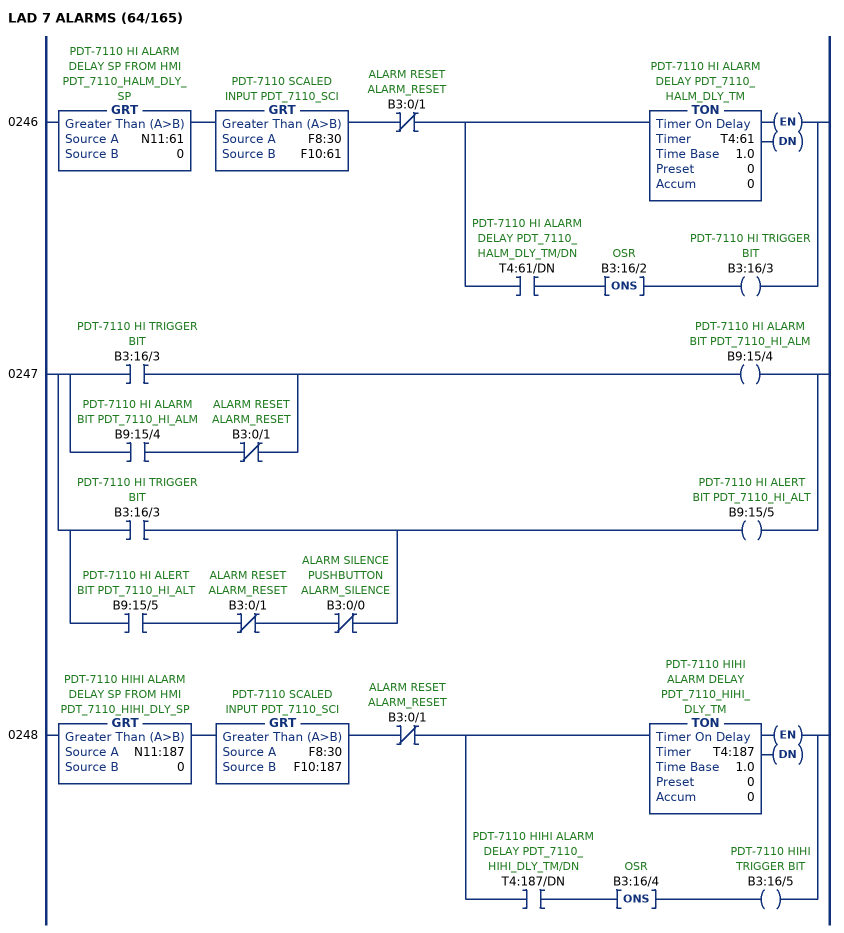
% Rung: 246 %
SOR GRT N11:61 0 GRT F8:30 F10:61 XIO B3:0/1 BST TON T4:61 1.0 0 0 NXB XIC T4:61/DN OSR B3:16/2 OTE B3:16/3 BND EOR
%   N11:61  PDT_7110_HALM_DLY_SP  "PDT-7110 HI ALARM DELAY SP FROM HMI" %
%   F8:30  PDT_7110_SCI  "PDT-7110 SCALED INPUT" %
%   F10:61  PDT_7110_HIALM_SP  "PDT-7110 HI ALARM SP" %
%   B3:0/1  ALARM_RESET  "ALARM RESET" %
%   T4:61  PDT_7110_HALM_DLY_TM  "PDT-7110 HI ALARM DELAY" %
%   B3:16/2  "OSR" %
%   B3:16/3  "PDT-7110 HI TRIGGER BIT" %
% Rung: 247 %
SOR BST BST XIC B3:16/3 NXB XIC B9:15/4 XIO B3:0/1 BND OTE B9:15/4 NXB BST XIC B3:16/3 NXB XIC B9:15/5 XIO B3:0/1 XIO B3:0/0 BND OTE B9:15/5 BND EOR
%   B3:16/3  "PDT-7110 HI TRIGGER BIT" %
%   B9:15/4  PDT_7110_HI_ALM  "PDT-7110 HI ALARM BIT" %
%   B3:0/1  ALARM_RESET  "ALARM RESET" %
%   B9:15/5  PDT_7110_HI_ALT  "PDT-7110 HI ALERT BIT" %
%   B3:0/0  ALARM_SILENCE  "ALARM SILENCE PUSHBUTTON" %
% Rung: 248 %
SOR GRT N11:187 0 GRT F8:30 F10:187 XIO B3:0/1 BST TON T4:187 1.0 0 0 NXB XIC T4:187/DN OSR B3:16/4 OTE B3:16/5 BND EOR
%   N11:187  PDT_7110_HIHI_DLY_SP  "PDT-7110 HIHI ALARM DELAY SP FROM HMI" %
%   F8:30  PDT_7110_SCI  "PDT-7110 SCALED INPUT" %
%   F10:187  PDT_7110_HIHI_SP  "PDT-7110 HIHI ALARM SP" %
%   B3:0/1  ALARM_RESET  "ALARM RESET" %
%   T4:187  PDT_7110_HIHI_DLY_TM  "PDT-7110 HIHI ALARM DELAY" %
%   B3:16/4  "OSR" %
%   B3:16/5  "PDT-7110 HIHI TRIGGER BIT" %

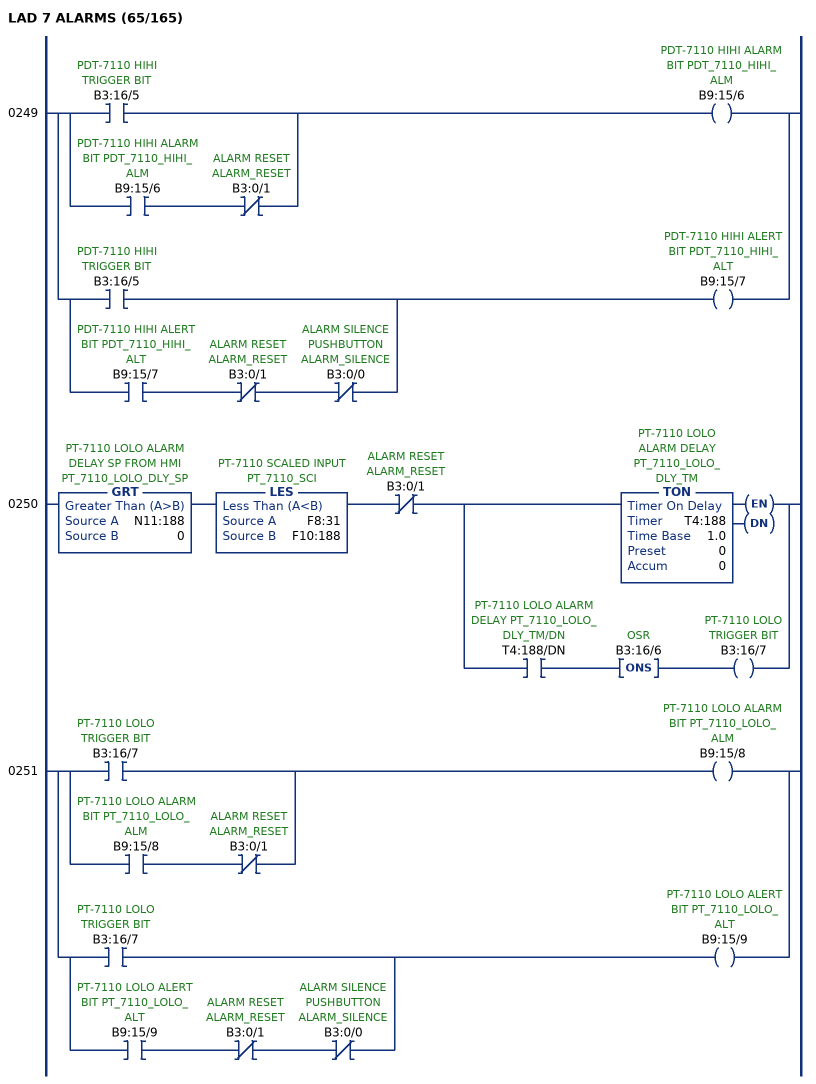
% Rung: 249 %
SOR BST BST XIC B3:16/5 NXB XIC B9:15/6 XIO B3:0/1 BND OTE B9:15/6 NXB BST XIC B3:16/5 NXB XIC B9:15/7 XIO B3:0/1 XIO B3:0/0 BND OTE B9:15/7 BND EOR
%   B3:16/5  "PDT-7110 HIHI TRIGGER BIT" %
%   B9:15/6  PDT_7110_HIHI_ALM  "PDT-7110 HIHI ALARM BIT" %
%   B3:0/1  ALARM_RESET  "ALARM RESET" %
%   B9:15/7  PDT_7110_HIHI_ALT  "PDT-7110 HIHI ALERT BIT" %
%   B3:0/0  ALARM_SILENCE  "ALARM SILENCE PUSHBUTTON" %
% Rung: 250 %
SOR GRT N11:188 0 LES F8:31 F10:188 XIO B3:0/1 BST TON T4:188 1.0 0 0 NXB XIC T4:188/DN OSR B3:16/6 OTE B3:16/7 BND EOR
%   N11:188  PT_7110_LOLO_DLY_SP  "PT-7110 LOLO ALARM DELAY SP FROM HMI" %
%   F8:31  PT_7110_SCI  "PT-7110 SCALED INPUT" %
%   F10:188  PT_7110_LOLO_SP  "PT-7110 LOLO ALARM SP" %
%   B3:0/1  ALARM_RESET  "ALARM RESET" %
%   T4:188  PT_7110_LOLO_DLY_TM  "PT-7110 LOLO ALARM DELAY" %
%   B3:16/6  "OSR" %
%   B3:16/7  "PT-7110 LOLO TRIGGER BIT" %
% Rung: 251 %
SOR BST BST XIC B3:16/7 NXB XIC B9:15/8 XIO B3:0/1 BND OTE B9:15/8 NXB BST XIC B3:16/7 NXB XIC B9:15/9 XIO B3:0/1 XIO B3:0/0 BND OTE B9:15/9 BND EOR
%   B3:16/7  "PT-7110 LOLO TRIGGER BIT" %
%   B9:15/8  PT_7110_LOLO_ALM  "PT-7110 LOLO ALARM BIT" %
%   B3:0/1  ALARM_RESET  "ALARM RESET" %
%   B9:15/9  PT_7110_LOLO_ALT  "PT-7110 LOLO ALERT BIT" %
%   B3:0/0  ALARM_SILENCE  "ALARM SILENCE PUSHBUTTON" %

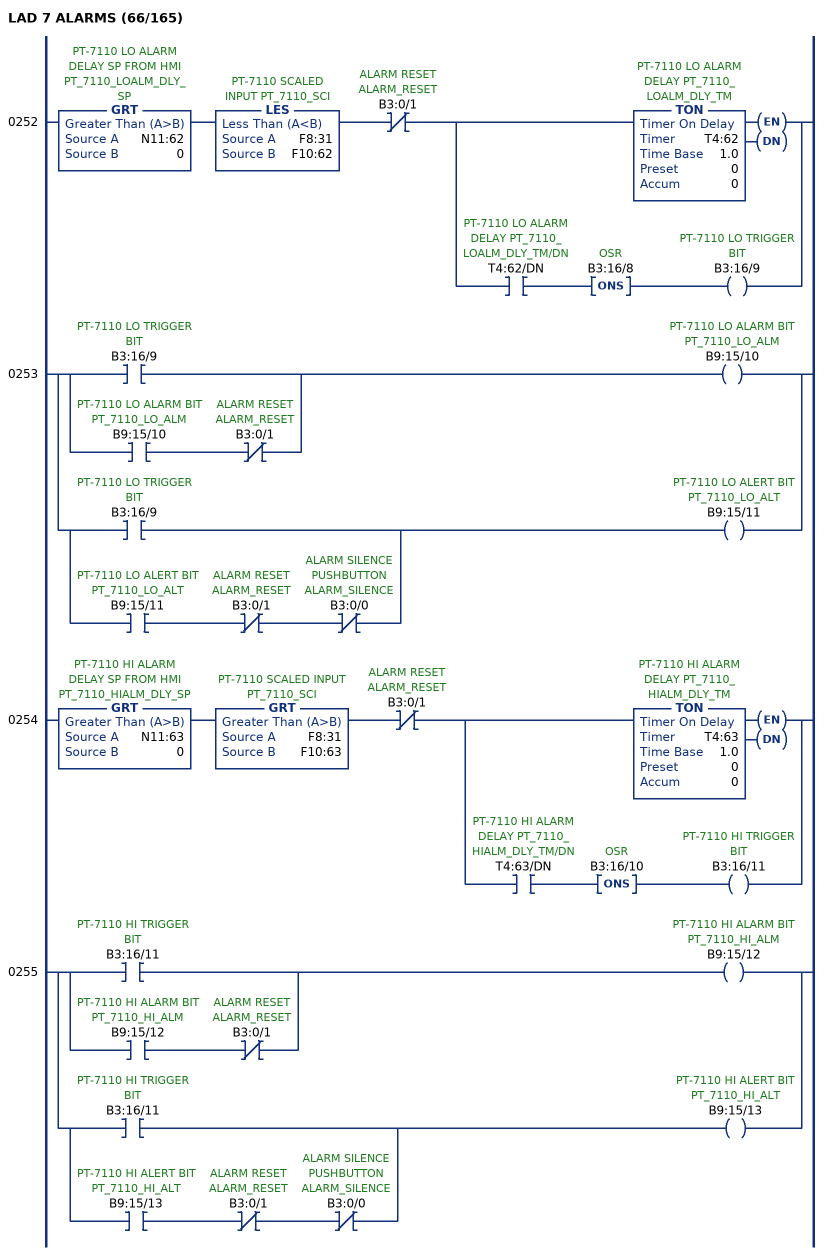
% Rung: 252 %
SOR GRT N11:62 0 LES F8:31 F10:62 XIO B3:0/1 BST TON T4:62 1.0 0 0 NXB XIC T4:62/DN OSR B3:16/8 OTE B3:16/9 BND EOR
%   N11:62  PT_7110_LOALM_DLY_SP  "PT-7110 LO ALARM DELAY SP FROM HMI" %
%   F8:31  PT_7110_SCI  "PT-7110 SCALED INPUT" %
%   F10:62  PT_7110_LOALM_SP  "PT-7110 LO ALARM SP" %
%   B3:0/1  ALARM_RESET  "ALARM RESET" %
%   T4:62  PT_7110_LOALM_DLY_TM  "PT-7110 LO ALARM DELAY" %
%   B3:16/8  "OSR" %
%   B3:16/9  "PT-7110 LO TRIGGER BIT" %
% Rung: 253 %
SOR BST BST XIC B3:16/9 NXB XIC B9:15/10 XIO B3:0/1 BND OTE B9:15/10 NXB BST XIC B3:16/9 NXB XIC B9:15/11 XIO B3:0/1 XIO B3:0/0 BND OTE B9:15/11 BND EOR
%   B3:16/9  "PT-7110 LO TRIGGER BIT" %
%   B9:15/10  PT_7110_LO_ALM  "PT-7110 LO ALARM BIT" %
%   B3:0/1  ALARM_RESET  "ALARM RESET" %
%   B9:15/11  PT_7110_LO_ALT  "PT-7110 LO ALERT BIT" %
%   B3:0/0  ALARM_SILENCE  "ALARM SILENCE PUSHBUTTON" %
% Rung: 254 %
SOR GRT N11:63 0 GRT F8:31 F10:63 XIO B3:0/1 BST TON T4:63 1.0 0 0 NXB XIC T4:63/DN OSR B3:16/10 OTE B3:16/11 BND EOR
%   N11:63  PT_7110_HIALM_DLY_SP  "PT-7110 HI ALARM DELAY SP FROM HMI" %
%   F8:31  PT_7110_SCI  "PT-7110 SCALED INPUT" %
%   F10:63  PT_7110_HIALM_SP  "PT-7110 HI ALARM SP" %
%   B3:0/1  ALARM_RESET  "ALARM RESET" %
%   T4:63  PT_7110_HIALM_DLY_TM  "PT-7110 HI ALARM DELAY" %
%   B3:16/10  "OSR" %
%   B3:16/11  "PT-7110 HI TRIGGER BIT" %
% Rung: 255 %
SOR BST BST XIC B3:16/11 NXB XIC B9:15/12 XIO B3:0/1 BND OTE B9:15/12 NXB BST XIC B3:16/11 NXB XIC B9:15/13 XIO B3:0/1 XIO B3:0/0 BND OTE B9:15/13 BND EOR
%   B3:16/11  "PT-7110 HI TRIGGER BIT" %
%   B9:15/12  PT_7110_HI_ALM  "PT-7110 HI ALARM BIT" %
%   B3:0/1  ALARM_RESET  "ALARM RESET" %
%   B9:15/13  PT_7110_HI_ALT  "PT-7110 HI ALERT BIT" %
%   B3:0/0  ALARM_SILENCE  "ALARM SILENCE PUSHBUTTON" %

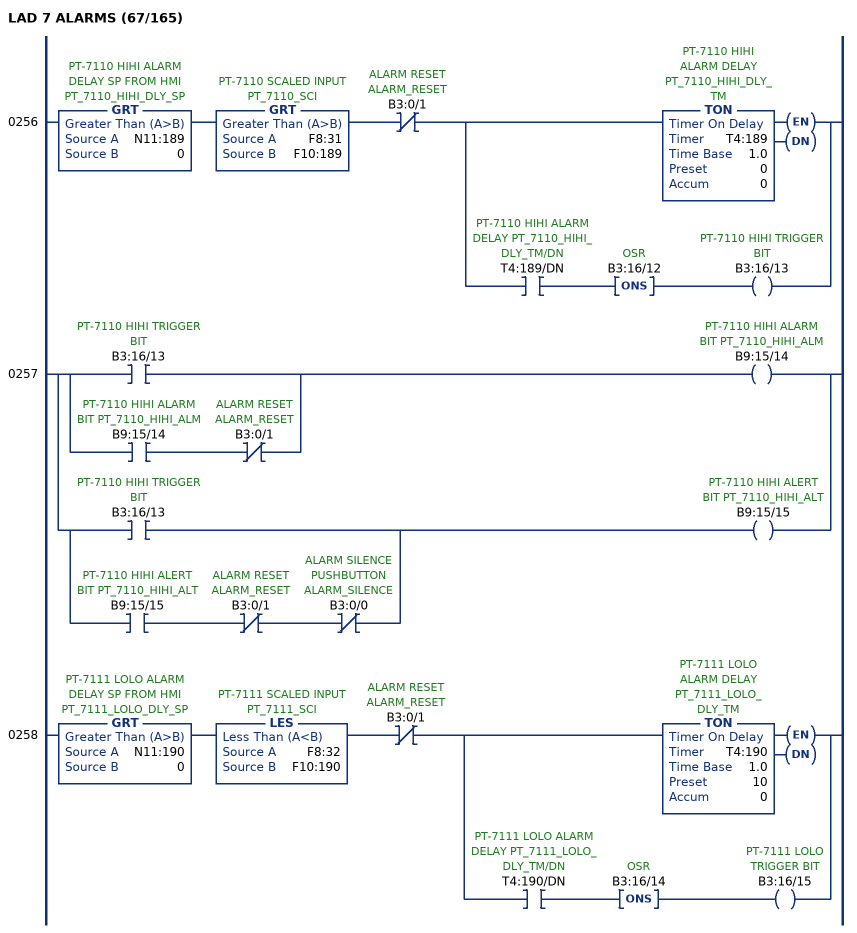
% Rung: 256 %
SOR GRT N11:189 0 GRT F8:31 F10:189 XIO B3:0/1 BST TON T4:189 1.0 0 0 NXB XIC T4:189/DN OSR B3:16/12 OTE B3:16/13 BND EOR
%   N11:189  PT_7110_HIHI_DLY_SP  "PT-7110 HIHI ALARM DELAY SP FROM HMI" %
%   F8:31  PT_7110_SCI  "PT-7110 SCALED INPUT" %
%   F10:189  PT_7110_HIHI_SP  "PT-7110 HIHI ALARM SP" %
%   B3:0/1  ALARM_RESET  "ALARM RESET" %
%   T4:189  PT_7110_HIHI_DLY_TM  "PT-7110 HIHI ALARM DELAY" %
%   B3:16/12  "OSR" %
%   B3:16/13  "PT-7110 HIHI TRIGGER BIT" %
% Rung: 257 %
SOR BST BST XIC B3:16/13 NXB XIC B9:15/14 XIO B3:0/1 BND OTE B9:15/14 NXB BST XIC B3:16/13 NXB XIC B9:15/15 XIO B3:0/1 XIO B3:0/0 BND OTE B9:15/15 BND EOR
%   B3:16/13  "PT-7110 HIHI TRIGGER BIT" %
%   B9:15/14  PT_7110_HIHI_ALM  "PT-7110 HIHI ALARM BIT" %
%   B3:0/1  ALARM_RESET  "ALARM RESET" %
%   B9:15/15  PT_7110_HIHI_ALT  "PT-7110 HIHI ALERT BIT" %
%   B3:0/0  ALARM_SILENCE  "ALARM SILENCE PUSHBUTTON" %
% Rung: 258 %
SOR GRT N11:190 0 LES F8:32 F10:190 XIO B3:0/1 BST TON T4:190 1.0 10 0 NXB XIC T4:190/DN OSR B3:16/14 OTE B3:16/15 BND EOR
%   N11:190  PT_7111_LOLO_DLY_SP  "PT-7111 LOLO ALARM DELAY SP FROM HMI" %
%   F8:32  PT_7111_SCI  "PT-7111 SCALED INPUT" %
%   F10:190  PT_7111_LOLO_SP  "PT-7111 LOLO ALARM SP" %
%   B3:0/1  ALARM_RESET  "ALARM RESET" %
%   T4:190  PT_7111_LOLO_DLY_TM  "PT-7111 LOLO ALARM DELAY" %
%   B3:16/14  "OSR" %
%   B3:16/15  "PT-7111 LOLO TRIGGER BIT" %

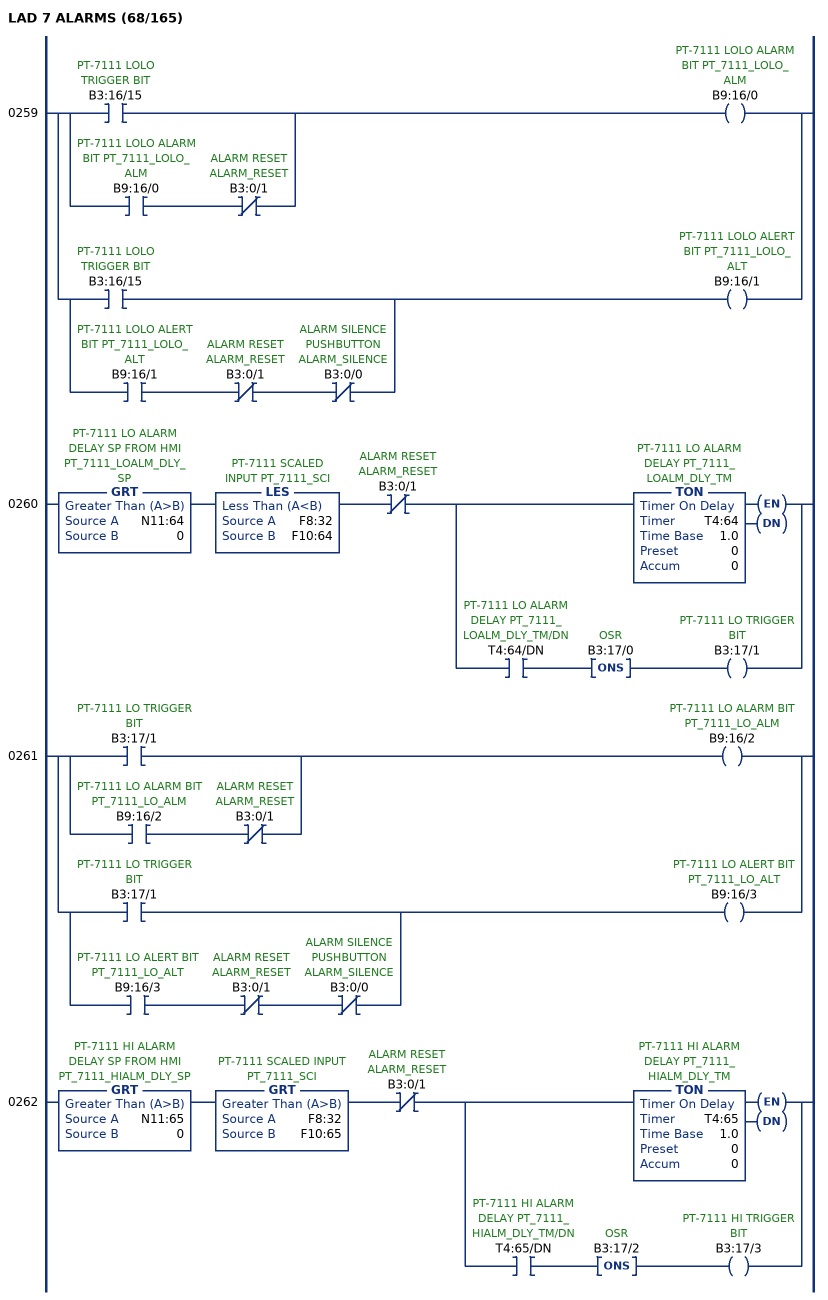
% Rung: 259 %
SOR BST BST XIC B3:16/15 NXB XIC B9:16/0 XIO B3:0/1 BND OTE B9:16/0 NXB BST XIC B3:16/15 NXB XIC B9:16/1 XIO B3:0/1 XIO B3:0/0 BND OTE B9:16/1 BND EOR
%   B3:16/15  "PT-7111 LOLO TRIGGER BIT" %
%   B9:16/0  PT_7111_LOLO_ALM  "PT-7111 LOLO ALARM BIT" %
%   B3:0/1  ALARM_RESET  "ALARM RESET" %
%   B9:16/1  PT_7111_LOLO_ALT  "PT-7111 LOLO ALERT BIT" %
%   B3:0/0  ALARM_SILENCE  "ALARM SILENCE PUSHBUTTON" %
% Rung: 260 %
SOR GRT N11:64 0 LES F8:32 F10:64 XIO B3:0/1 BST TON T4:64 1.0 0 0 NXB XIC T4:64/DN OSR B3:17/0 OTE B3:17/1 BND EOR
%   N11:64  PT_7111_LOALM_DLY_SP  "PT-7111 LO ALARM DELAY SP FROM HMI" %
%   F8:32  PT_7111_SCI  "PT-7111 SCALED INPUT" %
%   F10:64  PT_7111_LOALM_SP  "PT-7111 LO ALARM SP" %
%   B3:0/1  ALARM_RESET  "ALARM RESET" %
%   T4:64  PT_7111_LOALM_DLY_TM  "PT-7111 LO ALARM DELAY" %
%   B3:17/0  "OSR" %
%   B3:17/1  "PT-7111 LO TRIGGER BIT" %
% Rung: 261 %
SOR BST BST XIC B3:17/1 NXB XIC B9:16/2 XIO B3:0/1 BND OTE B9:16/2 NXB BST XIC B3:17/1 NXB XIC B9:16/3 XIO B3:0/1 XIO B3:0/0 BND OTE B9:16/3 BND EOR
%   B3:17/1  "PT-7111 LO TRIGGER BIT" %
%   B9:16/2  PT_7111_LO_ALM  "PT-7111 LO ALARM BIT" %
%   B3:0/1  ALARM_RESET  "ALARM RESET" %
%   B9:16/3  PT_7111_LO_ALT  "PT-7111 LO ALERT BIT" %
%   B3:0/0  ALARM_SILENCE  "ALARM SILENCE PUSHBUTTON" %
% Rung: 262 %
SOR GRT N11:65 0 GRT F8:32 F10:65 XIO B3:0/1 BST TON T4:65 1.0 0 0 NXB XIC T4:65/DN OSR B3:17/2 OTE B3:17/3 BND EOR
%   N11:65  PT_7111_HIALM_DLY_SP  "PT-7111 HI ALARM DELAY SP FROM HMI" %
%   F8:32  PT_7111_SCI  "PT-7111 SCALED INPUT" %
%   F10:65  PT_7111_HIALM_SP  "PT-7111 HI ALARM SP" %
%   B3:0/1  ALARM_RESET  "ALARM RESET" %
%   T4:65  PT_7111_HIALM_DLY_TM  "PT-7111 HI ALARM DELAY" %
%   B3:17/2  "OSR" %
%   B3:17/3  "PT-7111 HI TRIGGER BIT" %

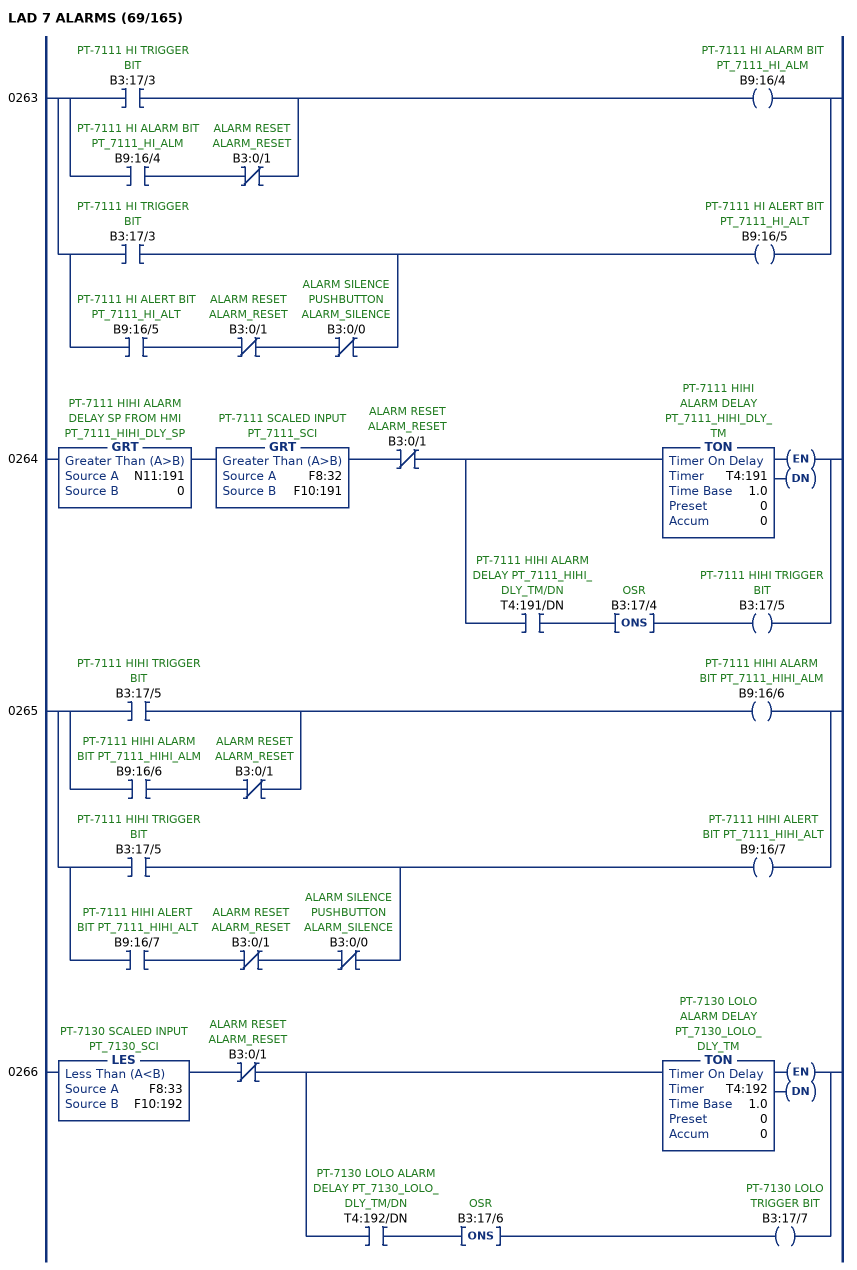
% Rung: 263 %
SOR BST BST XIC B3:17/3 NXB XIC B9:16/4 XIO B3:0/1 BND OTE B9:16/4 NXB BST XIC B3:17/3 NXB XIC B9:16/5 XIO B3:0/1 XIO B3:0/0 BND OTE B9:16/5 BND EOR
%   B3:17/3  "PT-7111 HI TRIGGER BIT" %
%   B9:16/4  PT_7111_HI_ALM  "PT-7111 HI ALARM BIT" %
%   B3:0/1  ALARM_RESET  "ALARM RESET" %
%   B9:16/5  PT_7111_HI_ALT  "PT-7111 HI ALERT BIT" %
%   B3:0/0  ALARM_SILENCE  "ALARM SILENCE PUSHBUTTON" %
% Rung: 264 %
SOR GRT N11:191 0 GRT F8:32 F10:191 XIO B3:0/1 BST TON T4:191 1.0 0 0 NXB XIC T4:191/DN OSR B3:17/4 OTE B3:17/5 BND EOR
%   N11:191  PT_7111_HIHI_DLY_SP  "PT-7111 HIHI ALARM DELAY SP FROM HMI" %
%   F8:32  PT_7111_SCI  "PT-7111 SCALED INPUT" %
%   F10:191  PT_7111_HIHI_SP  "PT-7111 HIHI ALARM SP" %
%   B3:0/1  ALARM_RESET  "ALARM RESET" %
%   T4:191  PT_7111_HIHI_DLY_TM  "PT-7111 HIHI ALARM DELAY" %
%   B3:17/4  "OSR" %
%   B3:17/5  "PT-7111 HIHI TRIGGER BIT" %
% Rung: 265 %
SOR BST BST XIC B3:17/5 NXB XIC B9:16/6 XIO B3:0/1 BND OTE B9:16/6 NXB BST XIC B3:17/5 NXB XIC B9:16/7 XIO B3:0/1 XIO B3:0/0 BND OTE B9:16/7 BND EOR
%   B3:17/5  "PT-7111 HIHI TRIGGER BIT" %
%   B9:16/6  PT_7111_HIHI_ALM  "PT-7111 HIHI ALARM BIT" %
%   B3:0/1  ALARM_RESET  "ALARM RESET" %
%   B9:16/7  PT_7111_HIHI_ALT  "PT-7111 HIHI ALERT BIT" %
%   B3:0/0  ALARM_SILENCE  "ALARM SILENCE PUSHBUTTON" %
% Rung: 266 %
SOR LES F8:33 F10:192 XIO B3:0/1 BST TON T4:192 1.0 0 0 NXB XIC T4:192/DN OSR B3:17/6 OTE B3:17/7 BND EOR
%   F8:33  PT_7130_SCI  "PT-7130 SCALED INPUT" %
%   F10:192  PT_7130_LOLO_SP  "PT-7130 LOLO ALARM SP" %
%   B3:0/1  ALARM_RESET  "ALARM RESET" %
%   T4:192  PT_7130_LOLO_DLY_TM  "PT-7130 LOLO ALARM DELAY" %
%   B3:17/6  "OSR" %
%   B3:17/7  "PT-7130 LOLO TRIGGER BIT" %

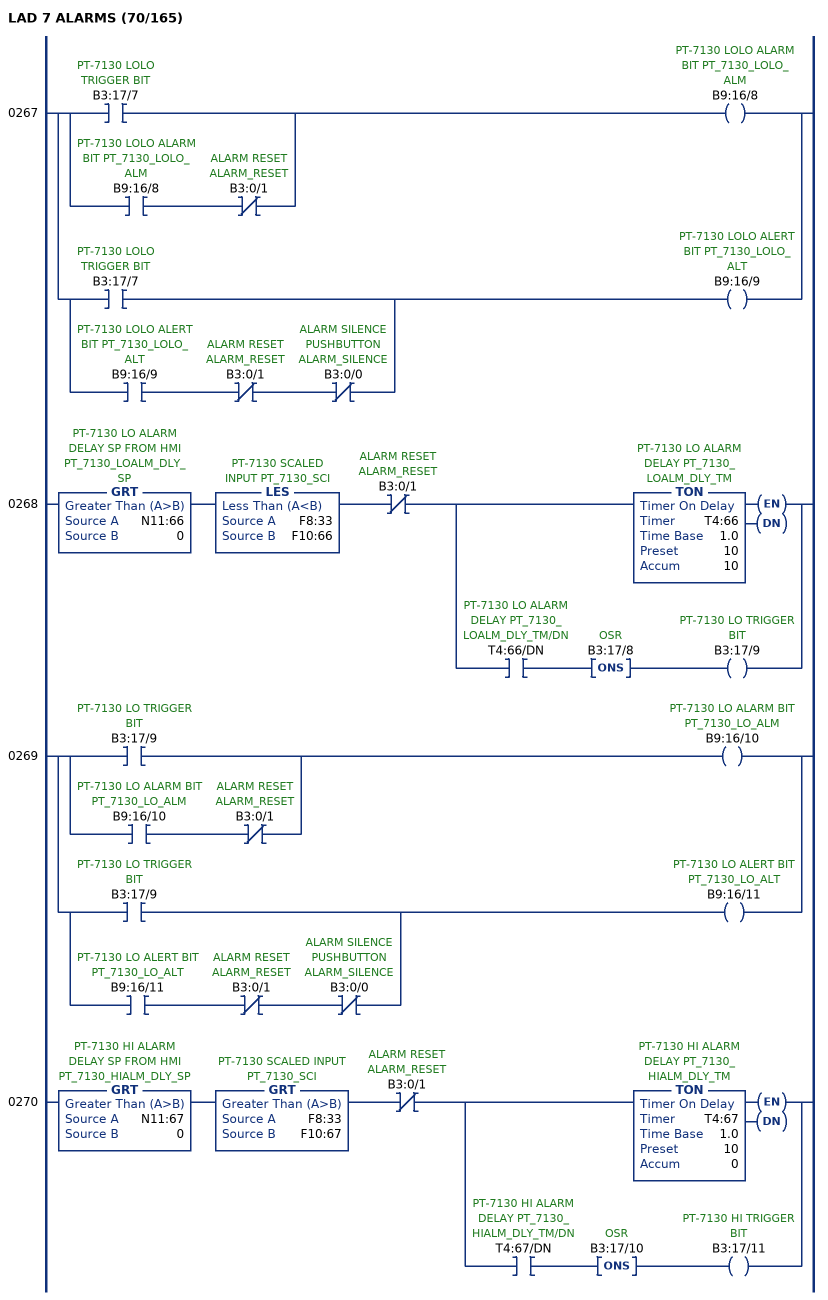
% Rung: 267 %
SOR BST BST XIC B3:17/7 NXB XIC B9:16/8 XIO B3:0/1 BND OTE B9:16/8 NXB BST XIC B3:17/7 NXB XIC B9:16/9 XIO B3:0/1 XIO B3:0/0 BND OTE B9:16/9 BND EOR
%   B3:17/7  "PT-7130 LOLO TRIGGER BIT" %
%   B9:16/8  PT_7130_LOLO_ALM  "PT-7130 LOLO ALARM BIT" %
%   B3:0/1  ALARM_RESET  "ALARM RESET" %
%   B9:16/9  PT_7130_LOLO_ALT  "PT-7130 LOLO ALERT BIT" %
%   B3:0/0  ALARM_SILENCE  "ALARM SILENCE PUSHBUTTON" %
% Rung: 268 %
SOR GRT N11:66 0 LES F8:33 F10:66 XIO B3:0/1 BST TON T4:66 1.0 10 10 NXB XIC T4:66/DN OSR B3:17/8 OTE B3:17/9 BND EOR
%   N11:66  PT_7130_LOALM_DLY_SP  "PT-7130 LO ALARM DELAY SP FROM HMI" %
%   F8:33  PT_7130_SCI  "PT-7130 SCALED INPUT" %
%   F10:66  PT_7130_LOALM_SP  "PT-7130 LO ALARM SP" %
%   B3:0/1  ALARM_RESET  "ALARM RESET" %
%   T4:66  PT_7130_LOALM_DLY_TM  "PT-7130 LO ALARM DELAY" %
%   B3:17/8  "OSR" %
%   B3:17/9  "PT-7130 LO TRIGGER BIT" %
% Rung: 269 %
SOR BST BST XIC B3:17/9 NXB XIC B9:16/10 XIO B3:0/1 BND OTE B9:16/10 NXB BST XIC B3:17/9 NXB XIC B9:16/11 XIO B3:0/1 XIO B3:0/0 BND OTE B9:16/11 BND EOR
%   B3:17/9  "PT-7130 LO TRIGGER BIT" %
%   B9:16/10  PT_7130_LO_ALM  "PT-7130 LO ALARM BIT" %
%   B3:0/1  ALARM_RESET  "ALARM RESET" %
%   B9:16/11  PT_7130_LO_ALT  "PT-7130 LO ALERT BIT" %
%   B3:0/0  ALARM_SILENCE  "ALARM SILENCE PUSHBUTTON" %
% Rung: 270 %
SOR GRT N11:67 0 GRT F8:33 F10:67 XIO B3:0/1 BST TON T4:67 1.0 10 0 NXB XIC T4:67/DN OSR B3:17/10 OTE B3:17/11 BND EOR
%   N11:67  PT_7130_HIALM_DLY_SP  "PT-7130 HI ALARM DELAY SP FROM HMI" %
%   F8:33  PT_7130_SCI  "PT-7130 SCALED INPUT" %
%   F10:67  PT_7130_HIALM_SP  "PT-7130 HI ALARM SP" %
%   B3:0/1  ALARM_RESET  "ALARM RESET" %
%   T4:67  PT_7130_HIALM_DLY_TM  "PT-7130 HI ALARM DELAY" %
%   B3:17/10  "OSR" %
%   B3:17/11  "PT-7130 HI TRIGGER BIT" %

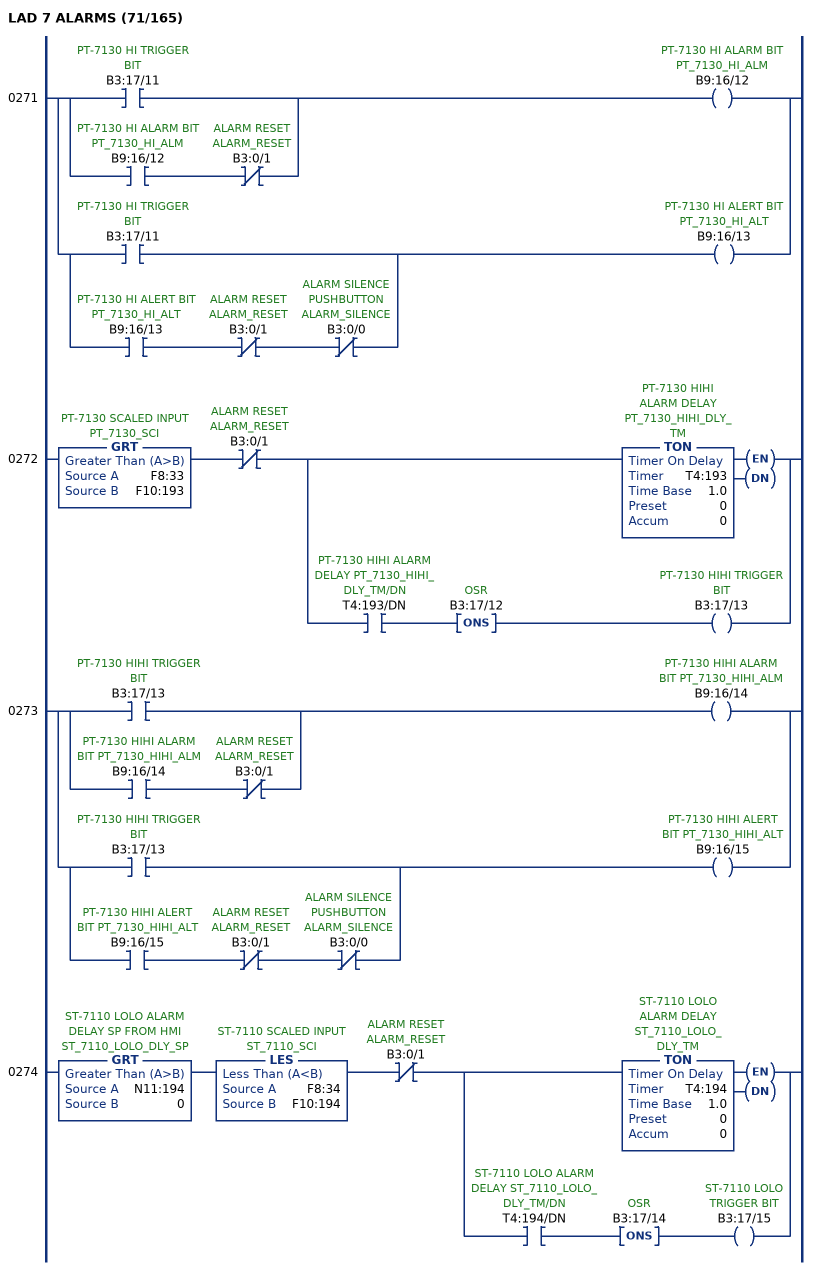
% Rung: 271 %
SOR BST BST XIC B3:17/11 NXB XIC B9:16/12 XIO B3:0/1 BND OTE B9:16/12 NXB BST XIC B3:17/11 NXB XIC B9:16/13 XIO B3:0/1 XIO B3:0/0 BND OTE B9:16/13 BND EOR
%   B3:17/11  "PT-7130 HI TRIGGER BIT" %
%   B9:16/12  PT_7130_HI_ALM  "PT-7130 HI ALARM BIT" %
%   B3:0/1  ALARM_RESET  "ALARM RESET" %
%   B9:16/13  PT_7130_HI_ALT  "PT-7130 HI ALERT BIT" %
%   B3:0/0  ALARM_SILENCE  "ALARM SILENCE PUSHBUTTON" %
% Rung: 272 %
SOR GRT F8:33 F10:193 XIO B3:0/1 BST TON T4:193 1.0 0 0 NXB XIC T4:193/DN OSR B3:17/12 OTE B3:17/13 BND EOR
%   F8:33  PT_7130_SCI  "PT-7130 SCALED INPUT" %
%   F10:193  PT_7130_HIHI_SP  "PT-7130 HIHI ALARM SP" %
%   B3:0/1  ALARM_RESET  "ALARM RESET" %
%   T4:193  PT_7130_HIHI_DLY_TM  "PT-7130 HIHI ALARM DELAY" %
%   B3:17/12  "OSR" %
%   B3:17/13  "PT-7130 HIHI TRIGGER BIT" %
% Rung: 273 %
SOR BST BST XIC B3:17/13 NXB XIC B9:16/14 XIO B3:0/1 BND OTE B9:16/14 NXB BST XIC B3:17/13 NXB XIC B9:16/15 XIO B3:0/1 XIO B3:0/0 BND OTE B9:16/15 BND EOR
%   B3:17/13  "PT-7130 HIHI TRIGGER BIT" %
%   B9:16/14  PT_7130_HIHI_ALM  "PT-7130 HIHI ALARM BIT" %
%   B3:0/1  ALARM_RESET  "ALARM RESET" %
%   B9:16/15  PT_7130_HIHI_ALT  "PT-7130 HIHI ALERT BIT" %
%   B3:0/0  ALARM_SILENCE  "ALARM SILENCE PUSHBUTTON" %
% Rung: 274 %
SOR GRT N11:194 0 LES F8:34 F10:194 XIO B3:0/1 BST TON T4:194 1.0 0 0 NXB XIC T4:194/DN OSR B3:17/14 OTE B3:17/15 BND EOR
%   N11:194  ST_7110_LOLO_DLY_SP  "ST-7110 LOLO ALARM DELAY SP FROM HMI" %
%   F8:34  ST_7110_SCI  "ST-7110 SCALED INPUT" %
%   F10:194  ST_7110_LOLO_SP  "ST-7110 LOLO ALARM SP" %
%   B3:0/1  ALARM_RESET  "ALARM RESET" %
%   T4:194  ST_7110_LOLO_DLY_TM  "ST-7110 LOLO ALARM DELAY" %
%   B3:17/14  "OSR" %
%   B3:17/15  "ST-7110 LOLO TRIGGER BIT" %

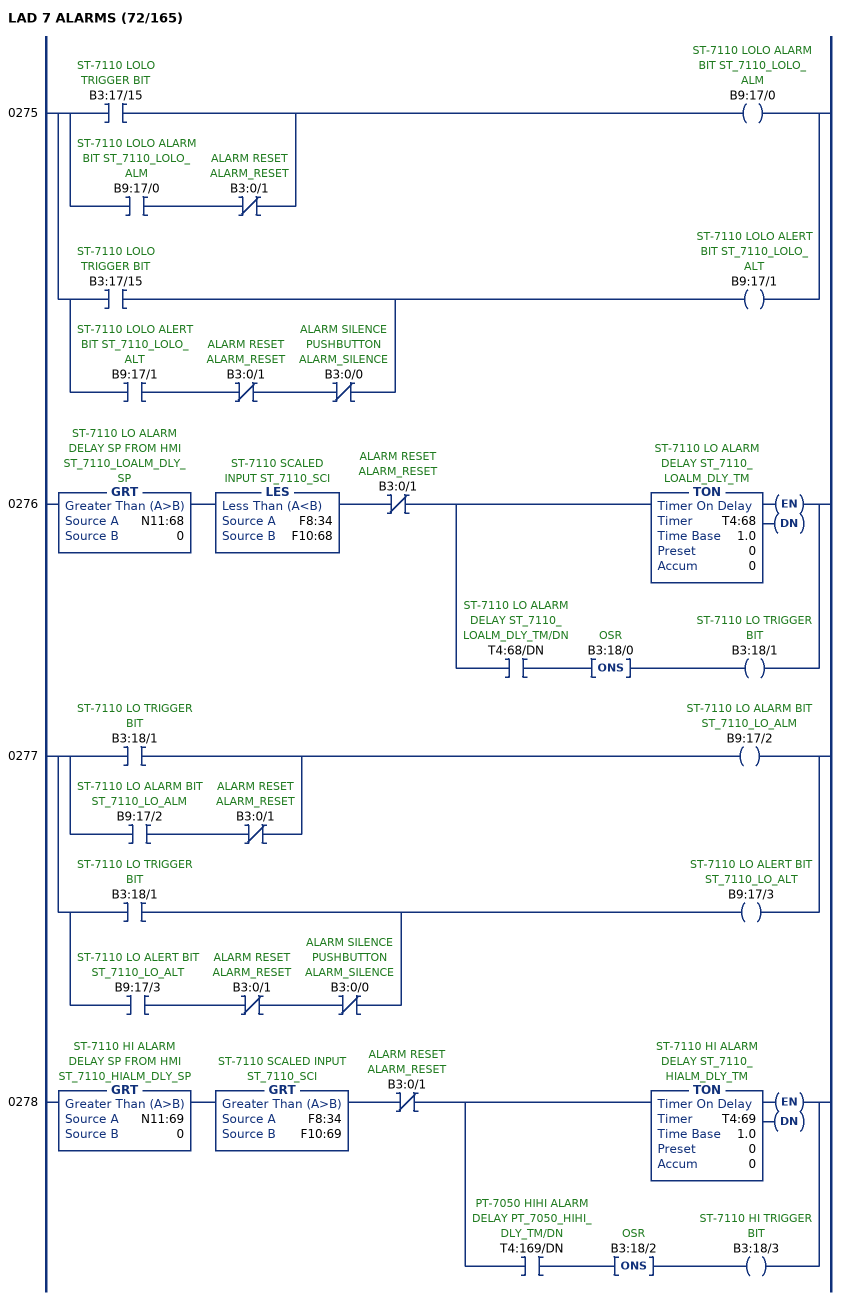
% Rung: 275 %
SOR BST BST XIC B3:17/15 NXB XIC B9:17/0 XIO B3:0/1 BND OTE B9:17/0 NXB BST XIC B3:17/15 NXB XIC B9:17/1 XIO B3:0/1 XIO B3:0/0 BND OTE B9:17/1 BND EOR
%   B3:17/15  "ST-7110 LOLO TRIGGER BIT" %
%   B9:17/0  ST_7110_LOLO_ALM  "ST-7110 LOLO ALARM BIT" %
%   B3:0/1  ALARM_RESET  "ALARM RESET" %
%   B9:17/1  ST_7110_LOLO_ALT  "ST-7110 LOLO ALERT BIT" %
%   B3:0/0  ALARM_SILENCE  "ALARM SILENCE PUSHBUTTON" %
% Rung: 276 %
SOR GRT N11:68 0 LES F8:34 F10:68 XIO B3:0/1 BST TON T4:68 1.0 0 0 NXB XIC T4:68/DN OSR B3:18/0 OTE B3:18/1 BND EOR
%   N11:68  ST_7110_LOALM_DLY_SP  "ST-7110 LO ALARM DELAY SP FROM HMI" %
%   F8:34  ST_7110_SCI  "ST-7110 SCALED INPUT" %
%   F10:68  ST_7110_LOALM_SP  "ST-7110 LO ALARM SP" %
%   B3:0/1  ALARM_RESET  "ALARM RESET" %
%   T4:68  ST_7110_LOALM_DLY_TM  "ST-7110 LO ALARM DELAY" %
%   B3:18/0  "OSR" %
%   B3:18/1  "ST-7110 LO TRIGGER BIT" %
% Rung: 277 %
SOR BST BST XIC B3:18/1 NXB XIC B9:17/2 XIO B3:0/1 BND OTE B9:17/2 NXB BST XIC B3:18/1 NXB XIC B9:17/3 XIO B3:0/1 XIO B3:0/0 BND OTE B9:17/3 BND EOR
%   B3:18/1  "ST-7110 LO TRIGGER BIT" %
%   B9:17/2  ST_7110_LO_ALM  "ST-7110 LO ALARM BIT" %
%   B3:0/1  ALARM_RESET  "ALARM RESET" %
%   B9:17/3  ST_7110_LO_ALT  "ST-7110 LO ALERT BIT" %
%   B3:0/0  ALARM_SILENCE  "ALARM SILENCE PUSHBUTTON" %
% Rung: 278 %
SOR GRT N11:69 0 GRT F8:34 F10:69 XIO B3:0/1 BST TON T4:69 1.0 0 0 NXB XIC T4:169/DN OSR B3:18/2 OTE B3:18/3 BND EOR
%   N11:69  ST_7110_HIALM_DLY_SP  "ST-7110 HI ALARM DELAY SP FROM HMI" %
%   F8:34  ST_7110_SCI  "ST-7110 SCALED INPUT" %
%   F10:69  ST_7110_HIALM_SP  "ST-7110 HI ALARM SP" %
%   B3:0/1  ALARM_RESET  "ALARM RESET" %
%   T4:69  ST_7110_HIALM_DLY_TM  "ST-7110 HI ALARM DELAY" %
%   T4:169  PT_7050_HIHI_DLY_TM  "PT-7050 HIHI ALARM DELAY" %
%   B3:18/2  "OSR" %
%   B3:18/3  "ST-7110 HI TRIGGER BIT" %

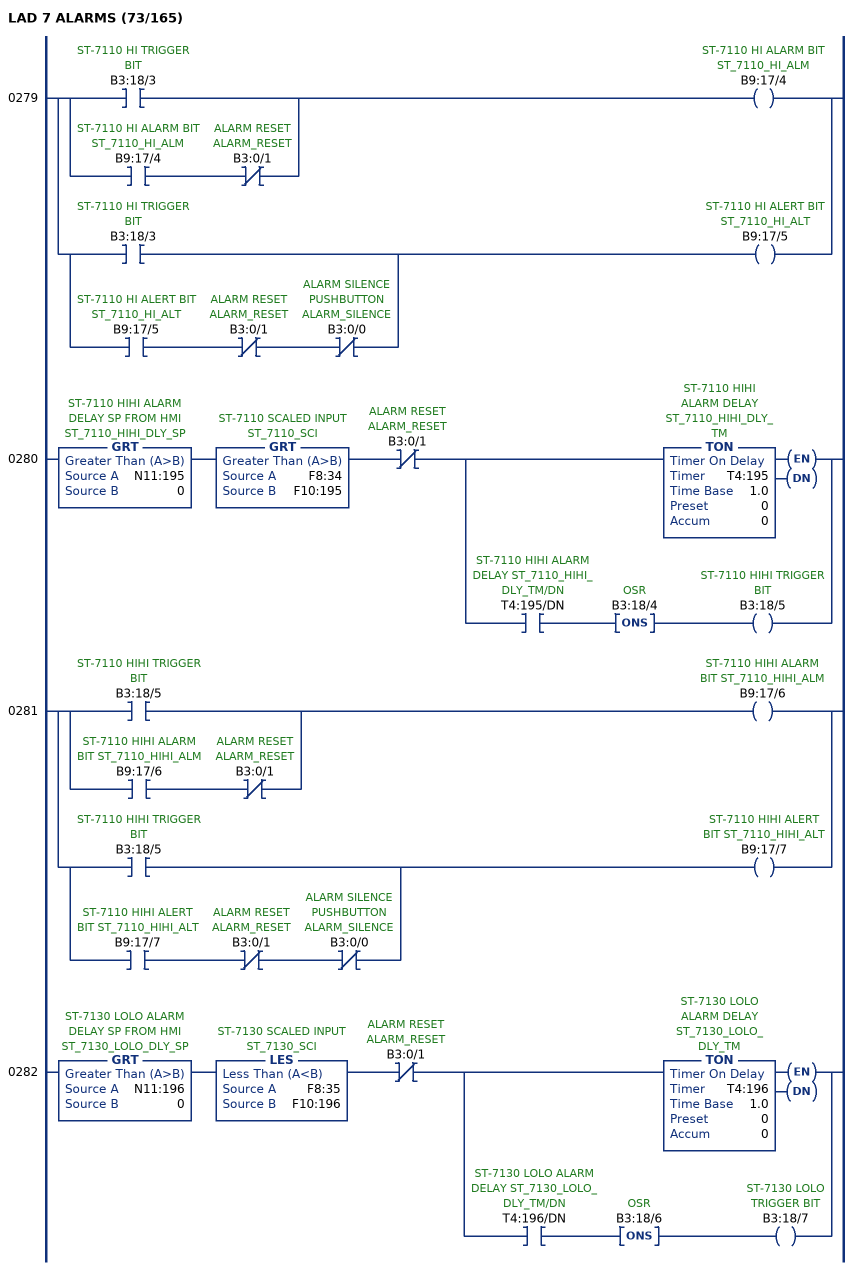
% Rung: 279 %
SOR BST BST XIC B3:18/3 NXB XIC B9:17/4 XIO B3:0/1 BND OTE B9:17/4 NXB BST XIC B3:18/3 NXB XIC B9:17/5 XIO B3:0/1 XIO B3:0/0 BND OTE B9:17/5 BND EOR
%   B3:18/3  "ST-7110 HI TRIGGER BIT" %
%   B9:17/4  ST_7110_HI_ALM  "ST-7110 HI ALARM BIT" %
%   B3:0/1  ALARM_RESET  "ALARM RESET" %
%   B9:17/5  ST_7110_HI_ALT  "ST-7110 HI ALERT BIT" %
%   B3:0/0  ALARM_SILENCE  "ALARM SILENCE PUSHBUTTON" %
% Rung: 280 %
SOR GRT N11:195 0 GRT F8:34 F10:195 XIO B3:0/1 BST TON T4:195 1.0 0 0 NXB XIC T4:195/DN OSR B3:18/4 OTE B3:18/5 BND EOR
%   N11:195  ST_7110_HIHI_DLY_SP  "ST-7110 HIHI ALARM DELAY SP FROM HMI" %
%   F8:34  ST_7110_SCI  "ST-7110 SCALED INPUT" %
%   F10:195  ST_7110_HIHI_SP  "ST-7110 HIHI ALARM SP" %
%   B3:0/1  ALARM_RESET  "ALARM RESET" %
%   T4:195  ST_7110_HIHI_DLY_TM  "ST-7110 HIHI ALARM DELAY" %
%   B3:18/4  "OSR" %
%   B3:18/5  "ST-7110 HIHI TRIGGER BIT" %
% Rung: 281 %
SOR BST BST XIC B3:18/5 NXB XIC B9:17/6 XIO B3:0/1 BND OTE B9:17/6 NXB BST XIC B3:18/5 NXB XIC B9:17/7 XIO B3:0/1 XIO B3:0/0 BND OTE B9:17/7 BND EOR
%   B3:18/5  "ST-7110 HIHI TRIGGER BIT" %
%   B9:17/6  ST_7110_HIHI_ALM  "ST-7110 HIHI ALARM BIT" %
%   B3:0/1  ALARM_RESET  "ALARM RESET" %
%   B9:17/7  ST_7110_HIHI_ALT  "ST-7110 HIHI ALERT BIT" %
%   B3:0/0  ALARM_SILENCE  "ALARM SILENCE PUSHBUTTON" %
% Rung: 282 %
SOR GRT N11:196 0 LES F8:35 F10:196 XIO B3:0/1 BST TON T4:196 1.0 0 0 NXB XIC T4:196/DN OSR B3:18/6 OTE B3:18/7 BND EOR
%   N11:196  ST_7130_LOLO_DLY_SP  "ST-7130 LOLO ALARM DELAY SP FROM HMI" %
%   F8:35  ST_7130_SCI  "ST-7130 SCALED INPUT" %
%   F10:196  ST_7130_LOLO_SP  "ST-7130 LOLO ALARM SP" %
%   B3:0/1  ALARM_RESET  "ALARM RESET" %
%   T4:196  ST_7130_LOLO_DLY_TM  "ST-7130 LOLO ALARM DELAY" %
%   B3:18/6  "OSR" %
%   B3:18/7  "ST-7130 LOLO TRIGGER BIT" %

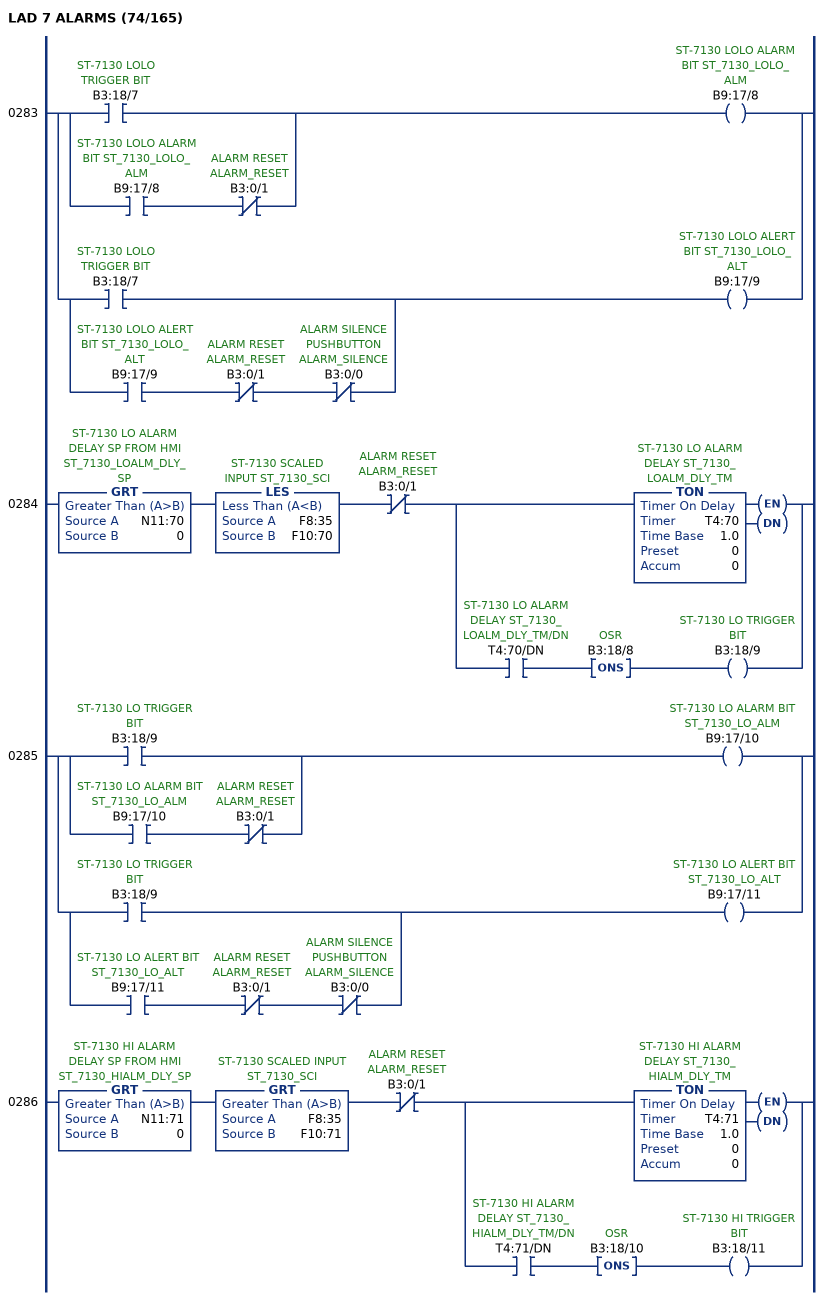
% Rung: 283 %
SOR BST BST XIC B3:18/7 NXB XIC B9:17/8 XIO B3:0/1 BND OTE B9:17/8 NXB BST XIC B3:18/7 NXB XIC B9:17/9 XIO B3:0/1 XIO B3:0/0 BND OTE B9:17/9 BND EOR
%   B3:18/7  "ST-7130 LOLO TRIGGER BIT" %
%   B9:17/8  ST_7130_LOLO_ALM  "ST-7130 LOLO ALARM BIT" %
%   B3:0/1  ALARM_RESET  "ALARM RESET" %
%   B9:17/9  ST_7130_LOLO_ALT  "ST-7130 LOLO ALERT BIT" %
%   B3:0/0  ALARM_SILENCE  "ALARM SILENCE PUSHBUTTON" %
% Rung: 284 %
SOR GRT N11:70 0 LES F8:35 F10:70 XIO B3:0/1 BST TON T4:70 1.0 0 0 NXB XIC T4:70/DN OSR B3:18/8 OTE B3:18/9 BND EOR
%   N11:70  ST_7130_LOALM_DLY_SP  "ST-7130 LO ALARM DELAY SP FROM HMI" %
%   F8:35  ST_7130_SCI  "ST-7130 SCALED INPUT" %
%   F10:70  ST_7130_LOALM_SP  "ST-7130 LO ALARM SP" %
%   B3:0/1  ALARM_RESET  "ALARM RESET" %
%   T4:70  ST_7130_LOALM_DLY_TM  "ST-7130 LO ALARM DELAY" %
%   B3:18/8  "OSR" %
%   B3:18/9  "ST-7130 LO TRIGGER BIT" %
% Rung: 285 %
SOR BST BST XIC B3:18/9 NXB XIC B9:17/10 XIO B3:0/1 BND OTE B9:17/10 NXB BST XIC B3:18/9 NXB XIC B9:17/11 XIO B3:0/1 XIO B3:0/0 BND OTE B9:17/11 BND EOR
%   B3:18/9  "ST-7130 LO TRIGGER BIT" %
%   B9:17/10  ST_7130_LO_ALM  "ST-7130 LO ALARM BIT" %
%   B3:0/1  ALARM_RESET  "ALARM RESET" %
%   B9:17/11  ST_7130_LO_ALT  "ST-7130 LO ALERT BIT" %
%   B3:0/0  ALARM_SILENCE  "ALARM SILENCE PUSHBUTTON" %
% Rung: 286 %
SOR GRT N11:71 0 GRT F8:35 F10:71 XIO B3:0/1 BST TON T4:71 1.0 0 0 NXB XIC T4:71/DN OSR B3:18/10 OTE B3:18/11 BND EOR
%   N11:71  ST_7130_HIALM_DLY_SP  "ST-7130 HI ALARM DELAY SP FROM HMI" %
%   F8:35  ST_7130_SCI  "ST-7130 SCALED INPUT" %
%   F10:71  ST_7130_HIALM_SP  "ST-7130 HI ALARM SP" %
%   B3:0/1  ALARM_RESET  "ALARM RESET" %
%   T4:71  ST_7130_HIALM_DLY_TM  "ST-7130 HI ALARM DELAY" %
%   B3:18/10  "OSR" %
%   B3:18/11  "ST-7130 HI TRIGGER BIT" %

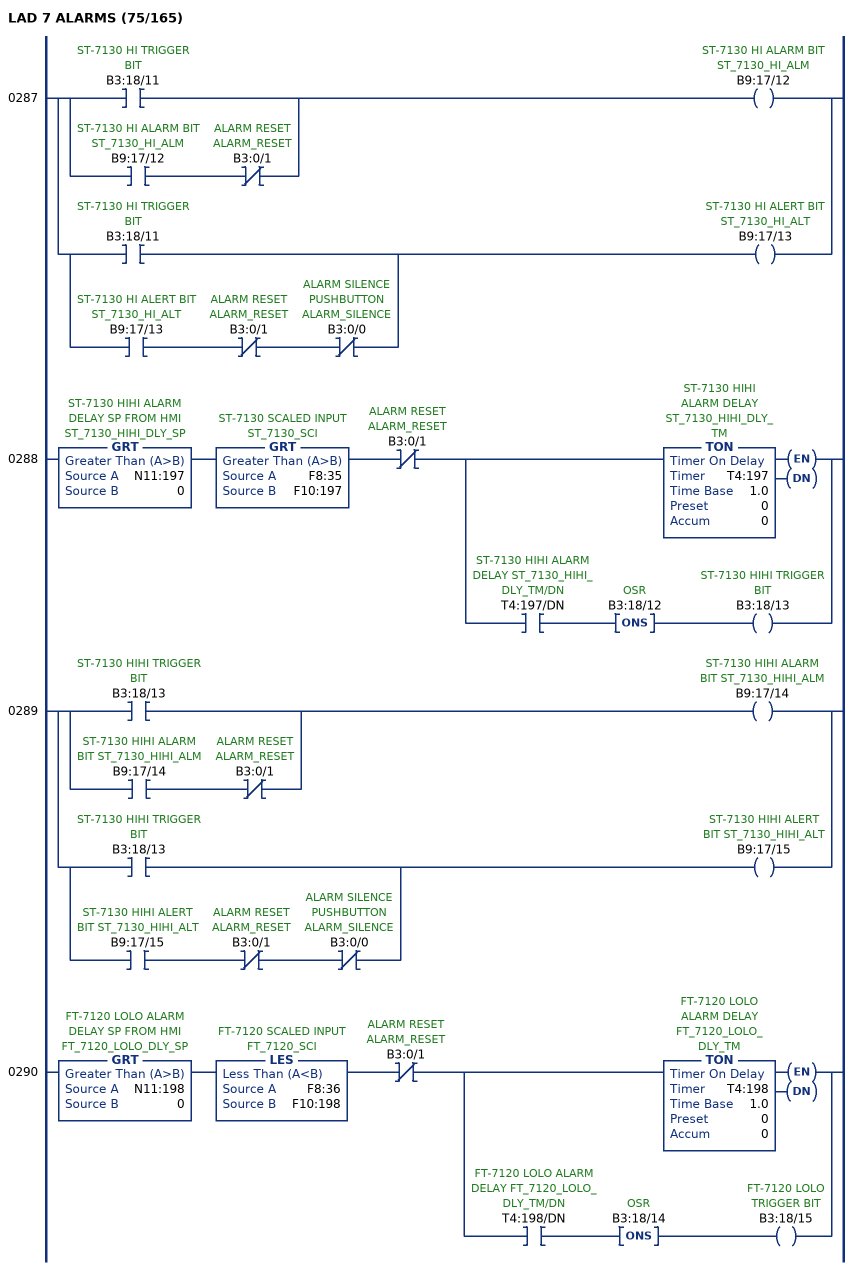
% Rung: 287 %
SOR BST BST XIC B3:18/11 NXB XIC B9:17/12 XIO B3:0/1 BND OTE B9:17/12 NXB BST XIC B3:18/11 NXB XIC B9:17/13 XIO B3:0/1 XIO B3:0/0 BND OTE B9:17/13 BND EOR
%   B3:18/11  "ST-7130 HI TRIGGER BIT" %
%   B9:17/12  ST_7130_HI_ALM  "ST-7130 HI ALARM BIT" %
%   B3:0/1  ALARM_RESET  "ALARM RESET" %
%   B9:17/13  ST_7130_HI_ALT  "ST-7130 HI ALERT BIT" %
%   B3:0/0  ALARM_SILENCE  "ALARM SILENCE PUSHBUTTON" %
% Rung: 288 %
SOR GRT N11:197 0 GRT F8:35 F10:197 XIO B3:0/1 BST TON T4:197 1.0 0 0 NXB XIC T4:197/DN OSR B3:18/12 OTE B3:18/13 BND EOR
%   N11:197  ST_7130_HIHI_DLY_SP  "ST-7130 HIHI ALARM DELAY SP FROM HMI" %
%   F8:35  ST_7130_SCI  "ST-7130 SCALED INPUT" %
%   F10:197  ST_7130_HIHI_SP  "ST-7130 HIHI ALARM SP" %
%   B3:0/1  ALARM_RESET  "ALARM RESET" %
%   T4:197  ST_7130_HIHI_DLY_TM  "ST-7130 HIHI ALARM DELAY" %
%   B3:18/12  "OSR" %
%   B3:18/13  "ST-7130 HIHI TRIGGER BIT" %
% Rung: 289 %
SOR BST BST XIC B3:18/13 NXB XIC B9:17/14 XIO B3:0/1 BND OTE B9:17/14 NXB BST XIC B3:18/13 NXB XIC B9:17/15 XIO B3:0/1 XIO B3:0/0 BND OTE B9:17/15 BND EOR
%   B3:18/13  "ST-7130 HIHI TRIGGER BIT" %
%   B9:17/14  ST_7130_HIHI_ALM  "ST-7130 HIHI ALARM BIT" %
%   B3:0/1  ALARM_RESET  "ALARM RESET" %
%   B9:17/15  ST_7130_HIHI_ALT  "ST-7130 HIHI ALERT BIT" %
%   B3:0/0  ALARM_SILENCE  "ALARM SILENCE PUSHBUTTON" %
% Rung: 290 %
SOR GRT N11:198 0 LES F8:36 F10:198 XIO B3:0/1 BST TON T4:198 1.0 0 0 NXB XIC T4:198/DN OSR B3:18/14 OTE B3:18/15 BND EOR
%   N11:198  FT_7120_LOLO_DLY_SP  "FT-7120 LOLO ALARM DELAY SP FROM HMI" %
%   F8:36  FT_7120_SCI  "FT-7120 SCALED INPUT" %
%   F10:198  FT_7120_LOLO_SP  "FT-7120 LOLO ALARM SP" %
%   B3:0/1  ALARM_RESET  "ALARM RESET" %
%   T4:198  FT_7120_LOLO_DLY_TM  "FT-7120 LOLO ALARM DELAY" %
%   B3:18/14  "OSR" %
%   B3:18/15  "FT-7120 LOLO TRIGGER BIT" %

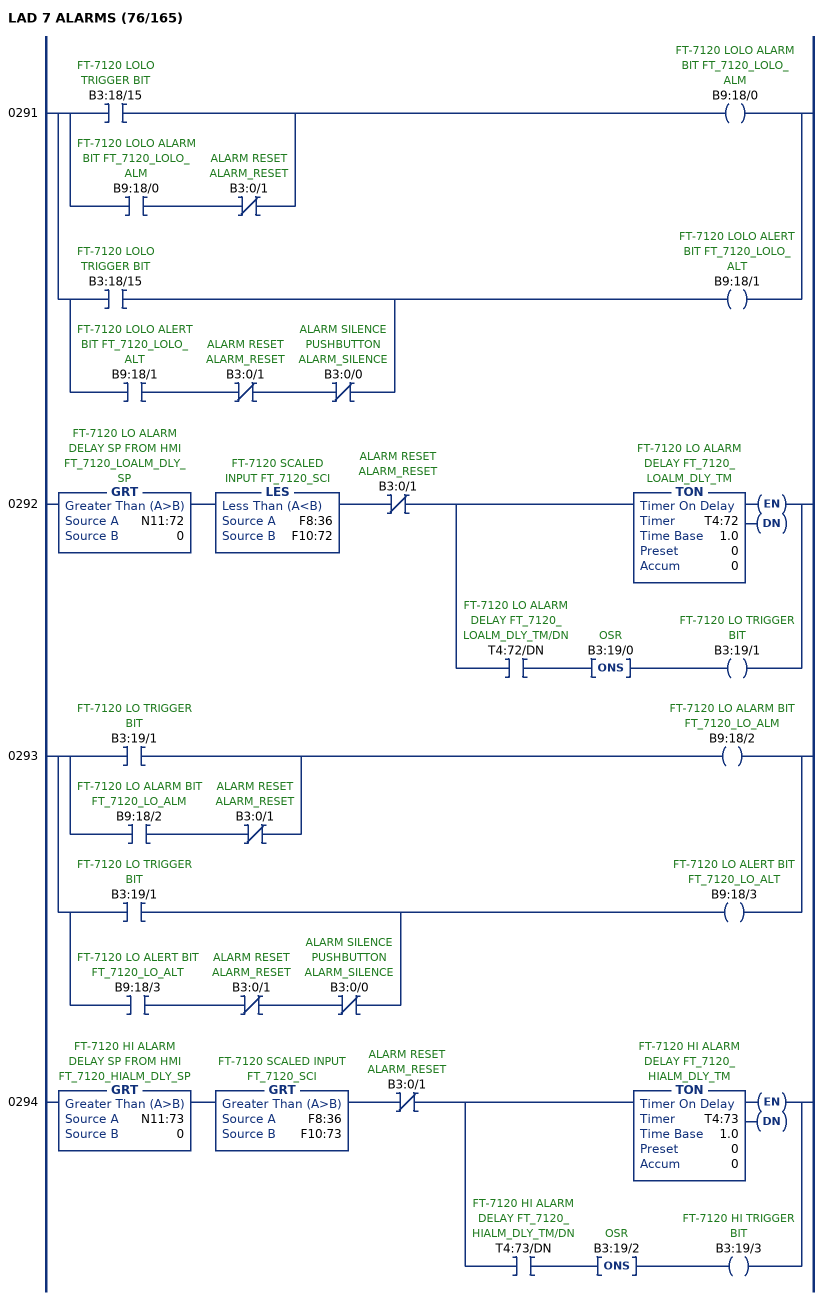
% Rung: 291 %
SOR BST BST XIC B3:18/15 NXB XIC B9:18/0 XIO B3:0/1 BND OTE B9:18/0 NXB BST XIC B3:18/15 NXB XIC B9:18/1 XIO B3:0/1 XIO B3:0/0 BND OTE B9:18/1 BND EOR
%   B3:18/15  "FT-7120 LOLO TRIGGER BIT" %
%   B9:18/0  FT_7120_LOLO_ALM  "FT-7120 LOLO ALARM BIT" %
%   B3:0/1  ALARM_RESET  "ALARM RESET" %
%   B9:18/1  FT_7120_LOLO_ALT  "FT-7120 LOLO ALERT BIT" %
%   B3:0/0  ALARM_SILENCE  "ALARM SILENCE PUSHBUTTON" %
% Rung: 292 %
SOR GRT N11:72 0 LES F8:36 F10:72 XIO B3:0/1 BST TON T4:72 1.0 0 0 NXB XIC T4:72/DN OSR B3:19/0 OTE B3:19/1 BND EOR
%   N11:72  FT_7120_LOALM_DLY_SP  "FT-7120 LO ALARM DELAY SP FROM HMI" %
%   F8:36  FT_7120_SCI  "FT-7120 SCALED INPUT" %
%   F10:72  FT_7120_LOALM_SP  "FT-7120 LO ALARM SP" %
%   B3:0/1  ALARM_RESET  "ALARM RESET" %
%   T4:72  FT_7120_LOALM_DLY_TM  "FT-7120 LO ALARM DELAY" %
%   B3:19/0  "OSR" %
%   B3:19/1  "FT-7120 LO TRIGGER BIT" %
% Rung: 293 %
SOR BST BST XIC B3:19/1 NXB XIC B9:18/2 XIO B3:0/1 BND OTE B9:18/2 NXB BST XIC B3:19/1 NXB XIC B9:18/3 XIO B3:0/1 XIO B3:0/0 BND OTE B9:18/3 BND EOR
%   B3:19/1  "FT-7120 LO TRIGGER BIT" %
%   B9:18/2  FT_7120_LO_ALM  "FT-7120 LO ALARM BIT" %
%   B3:0/1  ALARM_RESET  "ALARM RESET" %
%   B9:18/3  FT_7120_LO_ALT  "FT-7120 LO ALERT BIT" %
%   B3:0/0  ALARM_SILENCE  "ALARM SILENCE PUSHBUTTON" %
% Rung: 294 %
SOR GRT N11:73 0 GRT F8:36 F10:73 XIO B3:0/1 BST TON T4:73 1.0 0 0 NXB XIC T4:73/DN OSR B3:19/2 OTE B3:19/3 BND EOR
%   N11:73  FT_7120_HIALM_DLY_SP  "FT-7120 HI ALARM DELAY SP FROM HMI" %
%   F8:36  FT_7120_SCI  "FT-7120 SCALED INPUT" %
%   F10:73  FT_7120_HIALM_SP  "FT-7120 HI ALARM SP" %
%   B3:0/1  ALARM_RESET  "ALARM RESET" %
%   T4:73  FT_7120_HIALM_DLY_TM  "FT-7120 HI ALARM DELAY" %
%   B3:19/2  "OSR" %
%   B3:19/3  "FT-7120 HI TRIGGER BIT" %

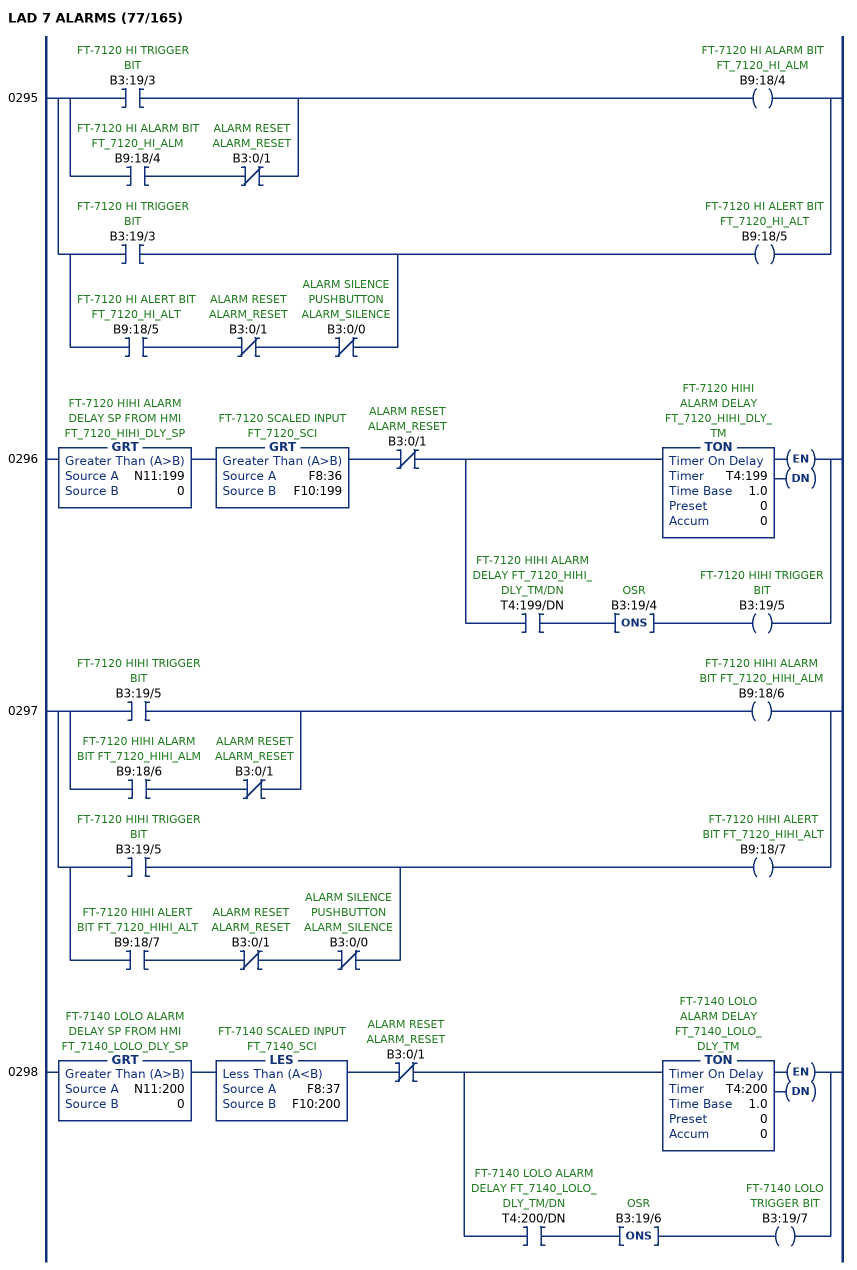
% Rung: 295 %
SOR BST BST XIC B3:19/3 NXB XIC B9:18/4 XIO B3:0/1 BND OTE B9:18/4 NXB BST XIC B3:19/3 NXB XIC B9:18/5 XIO B3:0/1 XIO B3:0/0 BND OTE B9:18/5 BND EOR
%   B3:19/3  "FT-7120 HI TRIGGER BIT" %
%   B9:18/4  FT_7120_HI_ALM  "FT-7120 HI ALARM BIT" %
%   B3:0/1  ALARM_RESET  "ALARM RESET" %
%   B9:18/5  FT_7120_HI_ALT  "FT-7120 HI ALERT BIT" %
%   B3:0/0  ALARM_SILENCE  "ALARM SILENCE PUSHBUTTON" %
% Rung: 296 %
SOR GRT N11:199 0 GRT F8:36 F10:199 XIO B3:0/1 BST TON T4:199 1.0 0 0 NXB XIC T4:199/DN OSR B3:19/4 OTE B3:19/5 BND EOR
%   N11:199  FT_7120_HIHI_DLY_SP  "FT-7120 HIHI ALARM DELAY SP FROM HMI" %
%   F8:36  FT_7120_SCI  "FT-7120 SCALED INPUT" %
%   F10:199  FT_7120_HIHI_SP  "FT-7120 HIHI ALARM SP" %
%   B3:0/1  ALARM_RESET  "ALARM RESET" %
%   T4:199  FT_7120_HIHI_DLY_TM  "FT-7120 HIHI ALARM DELAY" %
%   B3:19/4  "OSR" %
%   B3:19/5  "FT-7120 HIHI TRIGGER BIT" %
% Rung: 297 %
SOR BST BST XIC B3:19/5 NXB XIC B9:18/6 XIO B3:0/1 BND OTE B9:18/6 NXB BST XIC B3:19/5 NXB XIC B9:18/7 XIO B3:0/1 XIO B3:0/0 BND OTE B9:18/7 BND EOR
%   B3:19/5  "FT-7120 HIHI TRIGGER BIT" %
%   B9:18/6  FT_7120_HIHI_ALM  "FT-7120 HIHI ALARM BIT" %
%   B3:0/1  ALARM_RESET  "ALARM RESET" %
%   B9:18/7  FT_7120_HIHI_ALT  "FT-7120 HIHI ALERT BIT" %
%   B3:0/0  ALARM_SILENCE  "ALARM SILENCE PUSHBUTTON" %
% Rung: 298 %
SOR GRT N11:200 0 LES F8:37 F10:200 XIO B3:0/1 BST TON T4:200 1.0 0 0 NXB XIC T4:200/DN OSR B3:19/6 OTE B3:19/7 BND EOR
%   N11:200  FT_7140_LOLO_DLY_SP  "FT-7140 LOLO ALARM DELAY SP FROM HMI" %
%   F8:37  FT_7140_SCI  "FT-7140 SCALED INPUT" %
%   F10:200  FT_7140_LOLO_SP  "FT-7140 LOLO ALARM SP" %
%   B3:0/1  ALARM_RESET  "ALARM RESET" %
%   T4:200  FT_7140_LOLO_DLY_TM  "FT-7140 LOLO ALARM DELAY" %
%   B3:19/6  "OSR" %
%   B3:19/7  "FT-7140 LOLO TRIGGER BIT" %

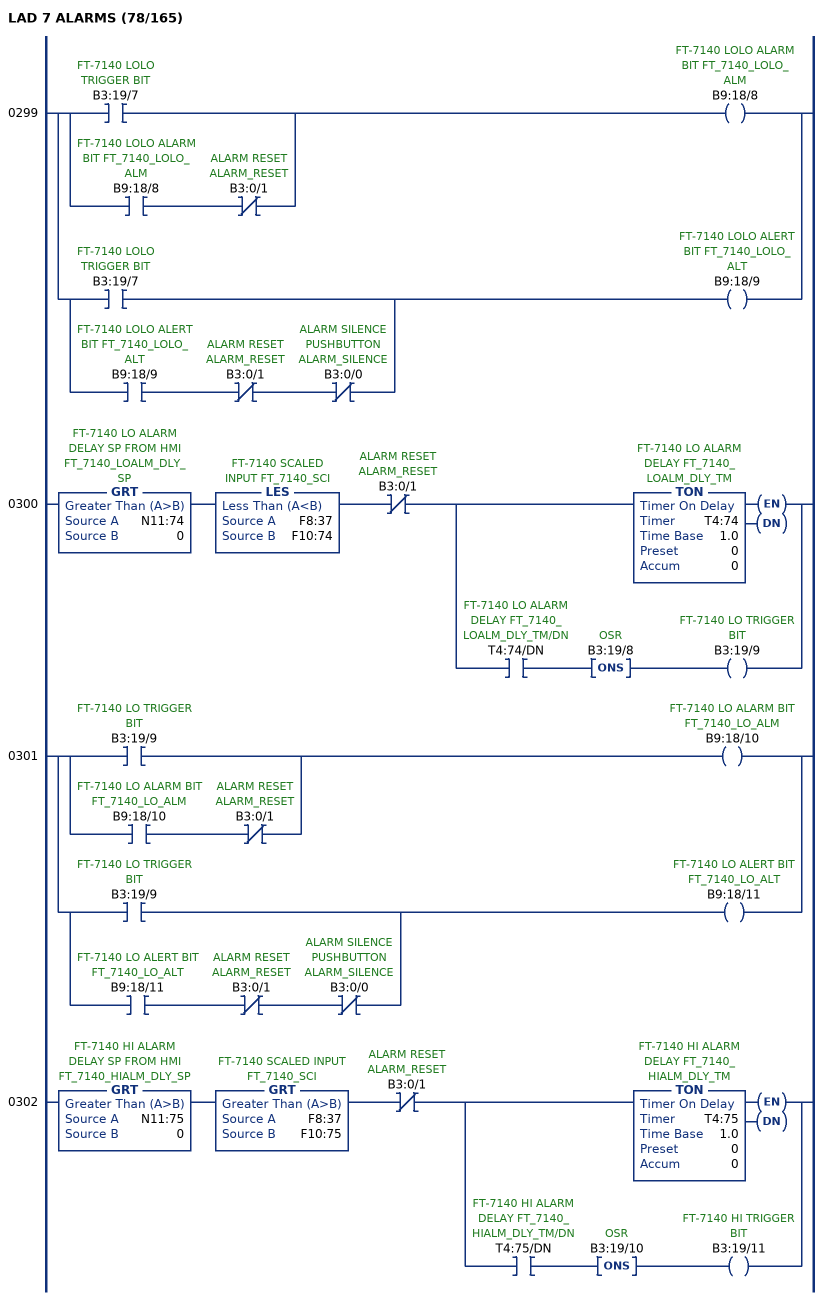
% Rung: 299 %
SOR BST BST XIC B3:19/7 NXB XIC B9:18/8 XIO B3:0/1 BND OTE B9:18/8 NXB BST XIC B3:19/7 NXB XIC B9:18/9 XIO B3:0/1 XIO B3:0/0 BND OTE B9:18/9 BND EOR
%   B3:19/7  "FT-7140 LOLO TRIGGER BIT" %
%   B9:18/8  FT_7140_LOLO_ALM  "FT-7140 LOLO ALARM BIT" %
%   B3:0/1  ALARM_RESET  "ALARM RESET" %
%   B9:18/9  FT_7140_LOLO_ALT  "FT-7140 LOLO ALERT BIT" %
%   B3:0/0  ALARM_SILENCE  "ALARM SILENCE PUSHBUTTON" %
% Rung: 300 %
SOR GRT N11:74 0 LES F8:37 F10:74 XIO B3:0/1 BST TON T4:74 1.0 0 0 NXB XIC T4:74/DN OSR B3:19/8 OTE B3:19/9 BND EOR
%   N11:74  FT_7140_LOALM_DLY_SP  "FT-7140 LO ALARM DELAY SP FROM HMI" %
%   F8:37  FT_7140_SCI  "FT-7140 SCALED INPUT" %
%   F10:74  FT_7140_LOALM_SP  "FT-7140 LO ALARM SP" %
%   B3:0/1  ALARM_RESET  "ALARM RESET" %
%   T4:74  FT_7140_LOALM_DLY_TM  "FT-7140 LO ALARM DELAY" %
%   B3:19/8  "OSR" %
%   B3:19/9  "FT-7140 LO TRIGGER BIT" %
% Rung: 301 %
SOR BST BST XIC B3:19/9 NXB XIC B9:18/10 XIO B3:0/1 BND OTE B9:18/10 NXB BST XIC B3:19/9 NXB XIC B9:18/11 XIO B3:0/1 XIO B3:0/0 BND OTE B9:18/11 BND EOR
%   B3:19/9  "FT-7140 LO TRIGGER BIT" %
%   B9:18/10  FT_7140_LO_ALM  "FT-7140 LO ALARM BIT" %
%   B3:0/1  ALARM_RESET  "ALARM RESET" %
%   B9:18/11  FT_7140_LO_ALT  "FT-7140 LO ALERT BIT" %
%   B3:0/0  ALARM_SILENCE  "ALARM SILENCE PUSHBUTTON" %
% Rung: 302 %
SOR GRT N11:75 0 GRT F8:37 F10:75 XIO B3:0/1 BST TON T4:75 1.0 0 0 NXB XIC T4:75/DN OSR B3:19/10 OTE B3:19/11 BND EOR
%   N11:75  FT_7140_HIALM_DLY_SP  "FT-7140 HI ALARM DELAY SP FROM HMI" %
%   F8:37  FT_7140_SCI  "FT-7140 SCALED INPUT" %
%   F10:75  FT_7140_HIALM_SP  "FT-7140 HI ALARM SP" %
%   B3:0/1  ALARM_RESET  "ALARM RESET" %
%   T4:75  FT_7140_HIALM_DLY_TM  "FT-7140 HI ALARM DELAY" %
%   B3:19/10  "OSR" %
%   B3:19/11  "FT-7140 HI TRIGGER BIT" %

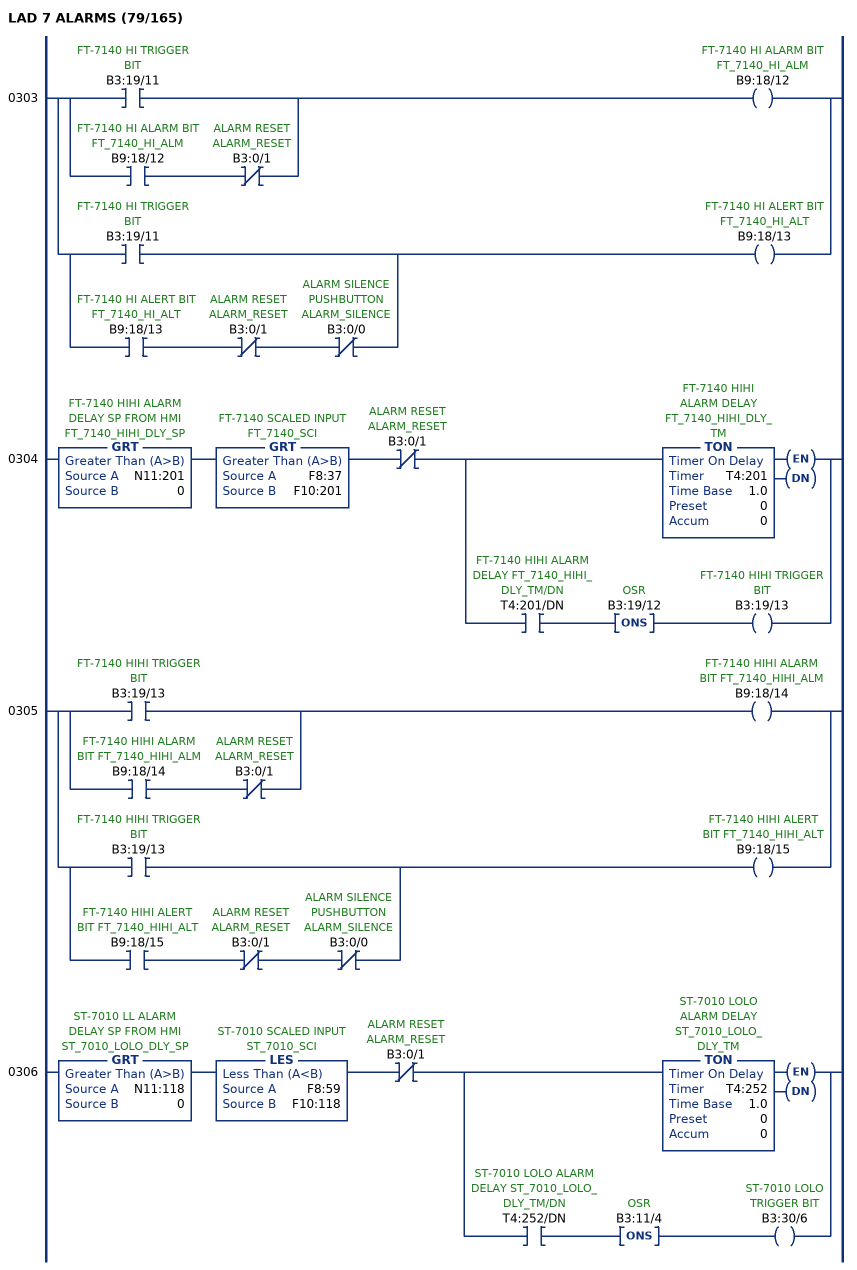
% Rung: 303 %
SOR BST BST XIC B3:19/11 NXB XIC B9:18/12 XIO B3:0/1 BND OTE B9:18/12 NXB BST XIC B3:19/11 NXB XIC B9:18/13 XIO B3:0/1 XIO B3:0/0 BND OTE B9:18/13 BND EOR
%   B3:19/11  "FT-7140 HI TRIGGER BIT" %
%   B9:18/12  FT_7140_HI_ALM  "FT-7140 HI ALARM BIT" %
%   B3:0/1  ALARM_RESET  "ALARM RESET" %
%   B9:18/13  FT_7140_HI_ALT  "FT-7140 HI ALERT BIT" %
%   B3:0/0  ALARM_SILENCE  "ALARM SILENCE PUSHBUTTON" %
% Rung: 304 %
SOR GRT N11:201 0 GRT F8:37 F10:201 XIO B3:0/1 BST TON T4:201 1.0 0 0 NXB XIC T4:201/DN OSR B3:19/12 OTE B3:19/13 BND EOR
%   N11:201  FT_7140_HIHI_DLY_SP  "FT-7140 HIHI ALARM DELAY SP FROM HMI" %
%   F8:37  FT_7140_SCI  "FT-7140 SCALED INPUT" %
%   F10:201  FT_7140_HIHI_SP  "FT-7140 HIHI ALARM SP" %
%   B3:0/1  ALARM_RESET  "ALARM RESET" %
%   T4:201  FT_7140_HIHI_DLY_TM  "FT-7140 HIHI ALARM DELAY" %
%   B3:19/12  "OSR" %
%   B3:19/13  "FT-7140 HIHI TRIGGER BIT" %
% Rung: 305 %
SOR BST BST XIC B3:19/13 NXB XIC B9:18/14 XIO B3:0/1 BND OTE B9:18/14 NXB BST XIC B3:19/13 NXB XIC B9:18/15 XIO B3:0/1 XIO B3:0/0 BND OTE B9:18/15 BND EOR
%   B3:19/13  "FT-7140 HIHI TRIGGER BIT" %
%   B9:18/14  FT_7140_HIHI_ALM  "FT-7140 HIHI ALARM BIT" %
%   B3:0/1  ALARM_RESET  "ALARM RESET" %
%   B9:18/15  FT_7140_HIHI_ALT  "FT-7140 HIHI ALERT BIT" %
%   B3:0/0  ALARM_SILENCE  "ALARM SILENCE PUSHBUTTON" %
% Rung: 306 %
SOR GRT N11:118 0 LES F8:59 F10:118 XIO B3:0/1 BST TON T4:252 1.0 0 0 NXB XIC T4:252/DN OSR B3:11/4 OTE B3:30/6 BND EOR
%   N11:118  ST_7010_LOLO_DLY_SP  "ST-7010 LL ALARM DELAY SP FROM HMI" %
%   F8:59  ST_7010_SCI  "ST-7010 SCALED INPUT" %
%   F10:118  ST_7010_LOLO_SP  "ST-7010 LOLO ALARM SP" %
%   B3:0/1  ALARM_RESET  "ALARM RESET" %
%   T4:252  ST_7010_LOLO_DLY_TM  "ST-7010 LOLO ALARM DELAY" %
%   B3:11/4  "OSR" %
%   B3:30/6  "ST-7010 LOLO TRIGGER BIT" %

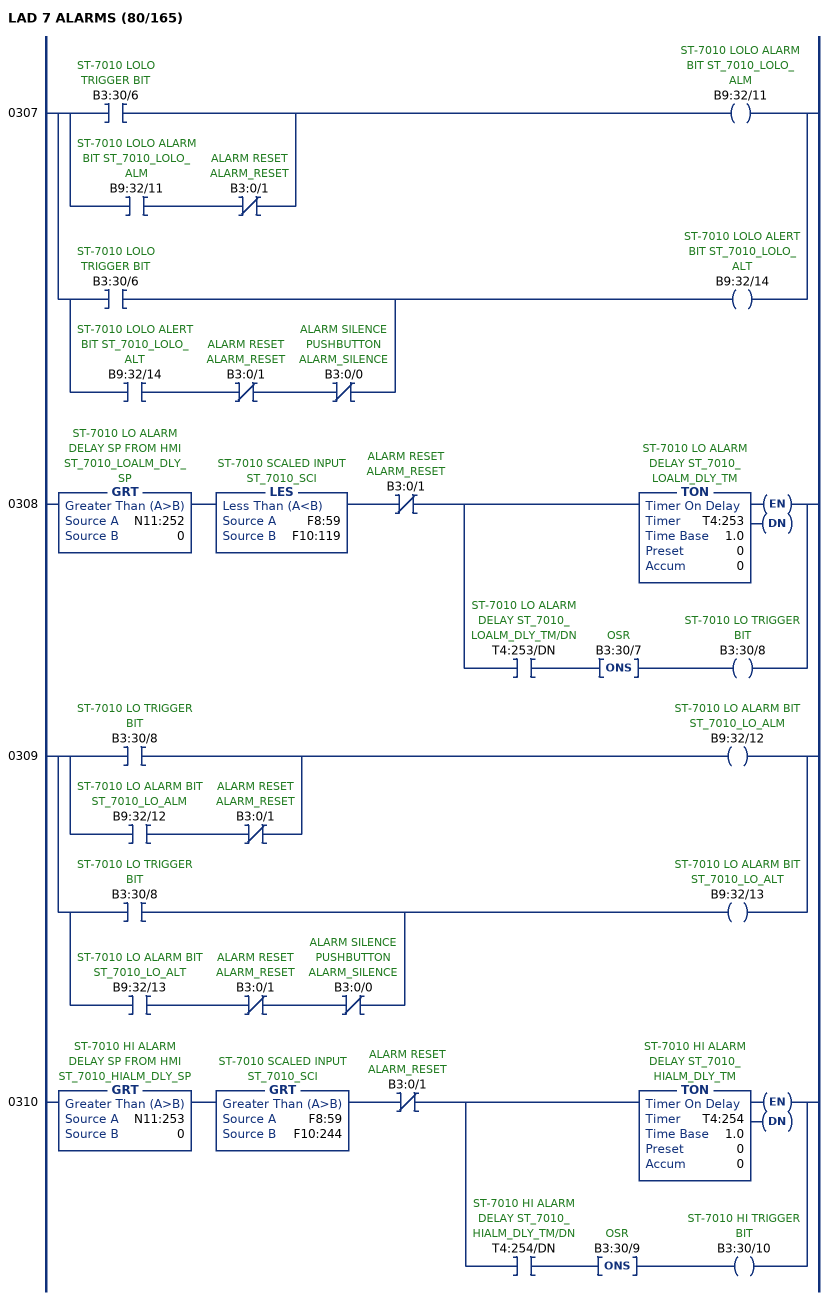
% Rung: 307 %
SOR BST BST XIC B3:30/6 NXB XIC B9:32/11 XIO B3:0/1 BND OTE B9:32/11 NXB BST XIC B3:30/6 NXB XIC B9:32/14 XIO B3:0/1 XIO B3:0/0 BND OTE B9:32/14 BND EOR
%   B3:30/6  "ST-7010 LOLO TRIGGER BIT" %
%   B9:32/11  ST_7010_LOLO_ALM  "ST-7010 LOLO ALARM BIT" %
%   B3:0/1  ALARM_RESET  "ALARM RESET" %
%   B9:32/14  ST_7010_LOLO_ALT  "ST-7010 LOLO ALERT BIT" %
%   B3:0/0  ALARM_SILENCE  "ALARM SILENCE PUSHBUTTON" %
% Rung: 308 %
SOR GRT N11:252 0 LES F8:59 F10:119 XIO B3:0/1 BST TON T4:253 1.0 0 0 NXB XIC T4:253/DN OSR B3:30/7 OTE B3:30/8 BND EOR
%   N11:252  ST_7010_LOALM_DLY_SP  "ST-7010 LO ALARM DELAY SP FROM HMI" %
%   F8:59  ST_7010_SCI  "ST-7010 SCALED INPUT" %
%   F10:119  ST_7010_LOALM_SP  "ST-7010 LO ALARM SP" %
%   B3:0/1  ALARM_RESET  "ALARM RESET" %
%   T4:253  ST_7010_LOALM_DLY_TM  "ST-7010 LO ALARM DELAY" %
%   B3:30/7  "OSR" %
%   B3:30/8  "ST-7010 LO TRIGGER BIT" %
% Rung: 309 %
SOR BST BST XIC B3:30/8 NXB XIC B9:32/12 XIO B3:0/1 BND OTE B9:32/12 NXB BST XIC B3:30/8 NXB XIC B9:32/13 XIO B3:0/1 XIO B3:0/0 BND OTE B9:32/13 BND EOR
%   B3:30/8  "ST-7010 LO TRIGGER BIT" %
%   B9:32/12  ST_7010_LO_ALM  "ST-7010 LO ALARM BIT" %
%   B3:0/1  ALARM_RESET  "ALARM RESET" %
%   B9:32/13  ST_7010_LO_ALT  "ST-7010 LO ALARM BIT" %
%   B3:0/0  ALARM_SILENCE  "ALARM SILENCE PUSHBUTTON" %
% Rung: 310 %
SOR GRT N11:253 0 GRT F8:59 F10:244 XIO B3:0/1 BST TON T4:254 1.0 0 0 NXB XIC T4:254/DN OSR B3:30/9 OTE B3:30/10 BND EOR
%   N11:253  ST_7010_HIALM_DLY_SP  "ST-7010 HI ALARM DELAY SP FROM HMI" %
%   F8:59  ST_7010_SCI  "ST-7010 SCALED INPUT" %
%   F10:244  ST_7010_HIALM_SP  "FT-7140 HI ALARM SP" %
%   B3:0/1  ALARM_RESET  "ALARM RESET" %
%   T4:254  ST_7010_HIALM_DLY_TM  "ST-7010 HI ALARM DELAY" %
%   B3:30/9  "OSR" %
%   B3:30/10  "ST-7010 HI TRIGGER BIT" %

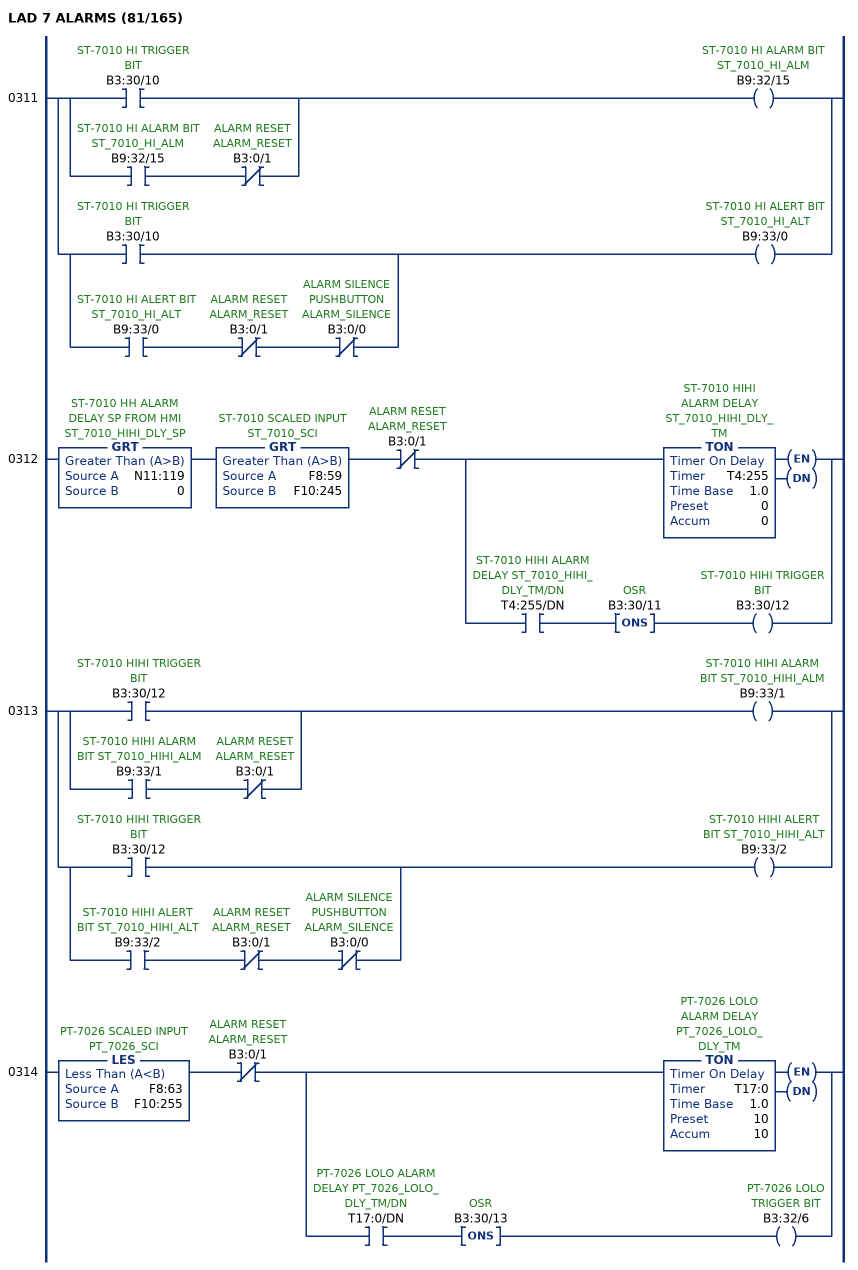
% Rung: 311 %
SOR BST BST XIC B3:30/10 NXB XIC B9:32/15 XIO B3:0/1 BND OTE B9:32/15 NXB BST XIC B3:30/10 NXB XIC B9:33/0 XIO B3:0/1 XIO B3:0/0 BND OTE B9:33/0 BND EOR
%   B3:30/10  "ST-7010 HI TRIGGER BIT" %
%   B9:32/15  ST_7010_HI_ALM  "ST-7010 HI ALARM BIT" %
%   B3:0/1  ALARM_RESET  "ALARM RESET" %
%   B9:33/0  ST_7010_HI_ALT  "ST-7010 HI ALERT BIT" %
%   B3:0/0  ALARM_SILENCE  "ALARM SILENCE PUSHBUTTON" %
% Rung: 312 %
SOR GRT N11:119 0 GRT F8:59 F10:245 XIO B3:0/1 BST TON T4:255 1.0 0 0 NXB XIC T4:255/DN OSR B3:30/11 OTE B3:30/12 BND EOR
%   N11:119  ST_7010_HIHI_DLY_SP  "ST-7010 HH ALARM DELAY SP FROM HMI" %
%   F8:59  ST_7010_SCI  "ST-7010 SCALED INPUT" %
%   F10:245  ST_7010_HIHI_SP  "ST-7010 HIHI ALARM SP" %
%   B3:0/1  ALARM_RESET  "ALARM RESET" %
%   T4:255  ST_7010_HIHI_DLY_TM  "ST-7010 HIHI ALARM DELAY" %
%   B3:30/11  "OSR" %
%   B3:30/12  "ST-7010 HIHI TRIGGER BIT" %
% Rung: 313 %
SOR BST BST XIC B3:30/12 NXB XIC B9:33/1 XIO B3:0/1 BND OTE B9:33/1 NXB BST XIC B3:30/12 NXB XIC B9:33/2 XIO B3:0/1 XIO B3:0/0 BND OTE B9:33/2 BND EOR
%   B3:30/12  "ST-7010 HIHI TRIGGER BIT" %
%   B9:33/1  ST_7010_HIHI_ALM  "ST-7010 HIHI ALARM BIT" %
%   B3:0/1  ALARM_RESET  "ALARM RESET" %
%   B9:33/2  ST_7010_HIHI_ALT  "ST-7010 HIHI ALERT BIT" %
%   B3:0/0  ALARM_SILENCE  "ALARM SILENCE PUSHBUTTON" %
% Rung: 314 %
SOR LES F8:63 F10:255 XIO B3:0/1 BST TON T17:0 1.0 10 10 NXB XIC T17:0/DN OSR B3:30/13 OTE B3:32/6 BND EOR
%   F8:63  PT_7026_SCI  "PT-7026 SCALED INPUT" %
%   F10:255  PT_7026_LOLO_SP  "PT-7026 LOLO ALARM SP" %
%   B3:0/1  ALARM_RESET  "ALARM RESET" %
%   T17:0  PT_7026_LOLO_DLY_TM  "PT-7026 LOLO ALARM DELAY" %
%   B3:30/13  "OSR" %
%   B3:32/6  "PT-7026 LOLO TRIGGER BIT" %

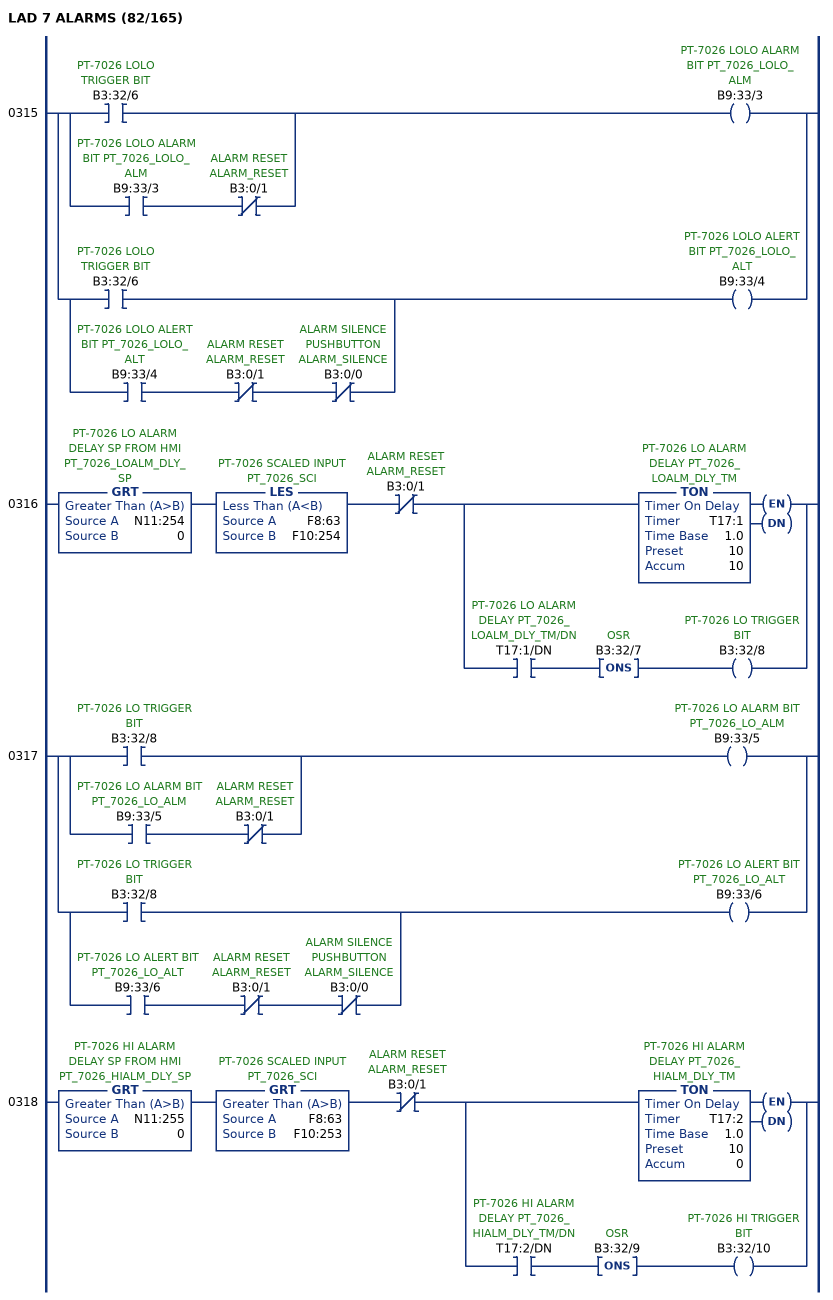
% Rung: 315 %
SOR BST BST XIC B3:32/6 NXB XIC B9:33/3 XIO B3:0/1 BND OTE B9:33/3 NXB BST XIC B3:32/6 NXB XIC B9:33/4 XIO B3:0/1 XIO B3:0/0 BND OTE B9:33/4 BND EOR
%   B3:32/6  "PT-7026 LOLO TRIGGER BIT" %
%   B9:33/3  PT_7026_LOLO_ALM  "PT-7026 LOLO ALARM BIT" %
%   B3:0/1  ALARM_RESET  "ALARM RESET" %
%   B9:33/4  PT_7026_LOLO_ALT  "PT-7026 LOLO ALERT BIT" %
%   B3:0/0  ALARM_SILENCE  "ALARM SILENCE PUSHBUTTON" %
% Rung: 316 %
SOR GRT N11:254 0 LES F8:63 F10:254 XIO B3:0/1 BST TON T17:1 1.0 10 10 NXB XIC T17:1/DN OSR B3:32/7 OTE B3:32/8 BND EOR
%   N11:254  PT_7026_LOALM_DLY_SP  "PT-7026 LO ALARM DELAY SP FROM HMI" %
%   F8:63  PT_7026_SCI  "PT-7026 SCALED INPUT" %
%   F10:254  PT_7026_LOALM_SP  "PT-7026 LO ALARM SP" %
%   B3:0/1  ALARM_RESET  "ALARM RESET" %
%   T17:1  PT_7026_LOALM_DLY_TM  "PT-7026 LO ALARM DELAY" %
%   B3:32/7  "OSR" %
%   B3:32/8  "PT-7026 LO TRIGGER BIT" %
% Rung: 317 %
SOR BST BST XIC B3:32/8 NXB XIC B9:33/5 XIO B3:0/1 BND OTE B9:33/5 NXB BST XIC B3:32/8 NXB XIC B9:33/6 XIO B3:0/1 XIO B3:0/0 BND OTE B9:33/6 BND EOR
%   B3:32/8  "PT-7026 LO TRIGGER BIT" %
%   B9:33/5  PT_7026_LO_ALM  "PT-7026 LO ALARM BIT" %
%   B3:0/1  ALARM_RESET  "ALARM RESET" %
%   B9:33/6  PT_7026_LO_ALT  "PT-7026 LO ALERT BIT" %
%   B3:0/0  ALARM_SILENCE  "ALARM SILENCE PUSHBUTTON" %
% Rung: 318 %
SOR GRT N11:255 0 GRT F8:63 F10:253 XIO B3:0/1 BST TON T17:2 1.0 10 0 NXB XIC T17:2/DN OSR B3:32/9 OTE B3:32/10 BND EOR
%   N11:255  PT_7026_HIALM_DLY_SP  "PT-7026 HI ALARM DELAY SP FROM HMI" %
%   F8:63  PT_7026_SCI  "PT-7026 SCALED INPUT" %
%   F10:253  PT_7026_HIALM_SP  "PT-7026 HI ALARM SP" %
%   B3:0/1  ALARM_RESET  "ALARM RESET" %
%   T17:2  PT_7026_HIALM_DLY_TM  "PT-7026 HI ALARM DELAY" %
%   B3:32/9  "OSR" %
%   B3:32/10  "PT-7026 HI TRIGGER BIT" %

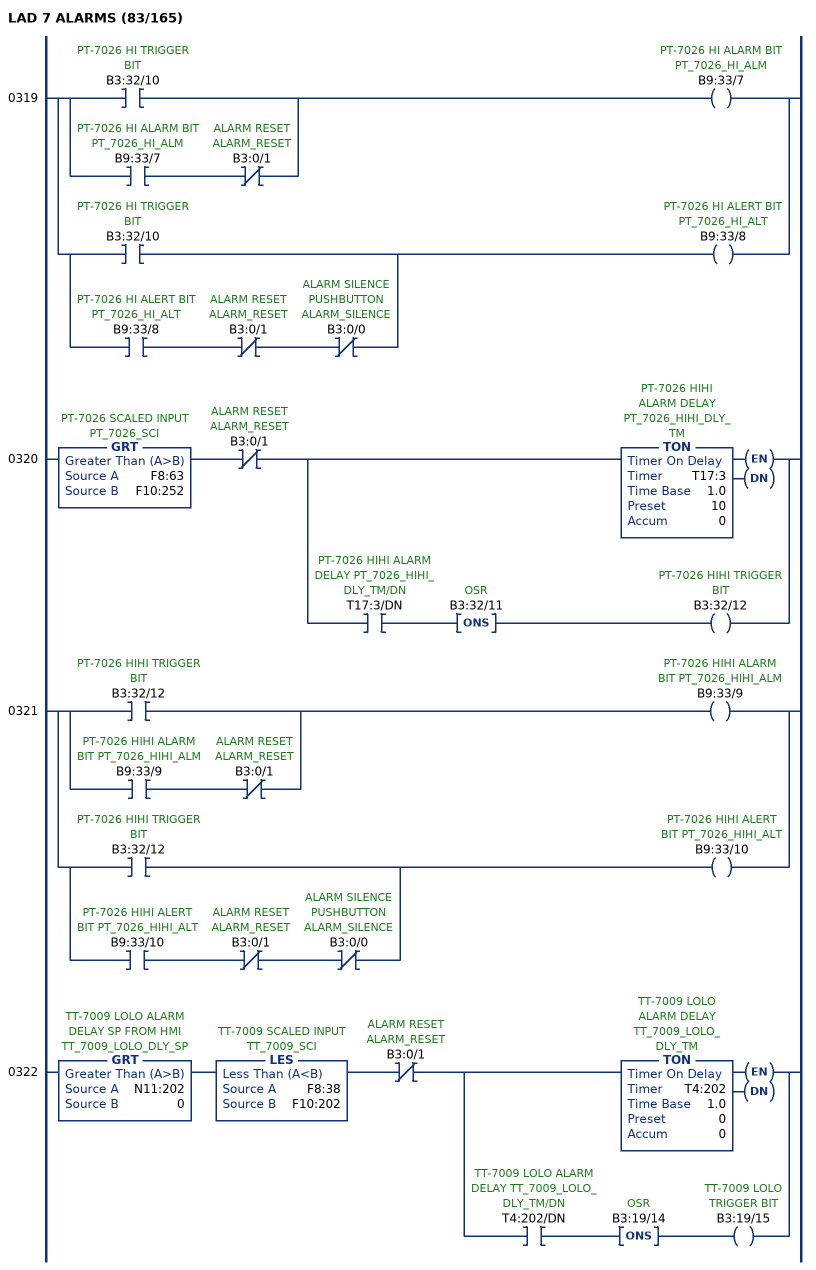
% Rung: 319 %
SOR BST BST XIC B3:32/10 NXB XIC B9:33/7 XIO B3:0/1 BND OTE B9:33/7 NXB BST XIC B3:32/10 NXB XIC B9:33/8 XIO B3:0/1 XIO B3:0/0 BND OTE B9:33/8 BND EOR
%   B3:32/10  "PT-7026 HI TRIGGER BIT" %
%   B9:33/7  PT_7026_HI_ALM  "PT-7026 HI ALARM BIT" %
%   B3:0/1  ALARM_RESET  "ALARM RESET" %
%   B9:33/8  PT_7026_HI_ALT  "PT-7026 HI ALERT BIT" %
%   B3:0/0  ALARM_SILENCE  "ALARM SILENCE PUSHBUTTON" %
% Rung: 320 %
SOR GRT F8:63 F10:252 XIO B3:0/1 BST TON T17:3 1.0 10 0 NXB XIC T17:3/DN OSR B3:32/11 OTE B3:32/12 BND EOR
%   F8:63  PT_7026_SCI  "PT-7026 SCALED INPUT" %
%   F10:252  PT_7026_HIHI_SP  "PT-7026 HIHI ALARM SP" %
%   B3:0/1  ALARM_RESET  "ALARM RESET" %
%   T17:3  PT_7026_HIHI_DLY_TM  "PT-7026 HIHI ALARM DELAY" %
%   B3:32/11  "OSR" %
%   B3:32/12  "PT-7026 HIHI TRIGGER BIT" %
% Rung: 321 %
SOR BST BST XIC B3:32/12 NXB XIC B9:33/9 XIO B3:0/1 BND OTE B9:33/9 NXB BST XIC B3:32/12 NXB XIC B9:33/10 XIO B3:0/1 XIO B3:0/0 BND OTE B9:33/10 BND EOR
%   B3:32/12  "PT-7026 HIHI TRIGGER BIT" %
%   B9:33/9  PT_7026_HIHI_ALM  "PT-7026 HIHI ALARM BIT" %
%   B3:0/1  ALARM_RESET  "ALARM RESET" %
%   B9:33/10  PT_7026_HIHI_ALT  "PT-7026 HIHI ALERT BIT" %
%   B3:0/0  ALARM_SILENCE  "ALARM SILENCE PUSHBUTTON" %
% Rung: 322 %
SOR GRT N11:202 0 LES F8:38 F10:202 XIO B3:0/1 BST TON T4:202 1.0 0 0 NXB XIC T4:202/DN OSR B3:19/14 OTE B3:19/15 BND EOR
%   N11:202  TT_7009_LOLO_DLY_SP  "TT-7009 LOLO ALARM DELAY SP FROM HMI" %
%   F8:38  TT_7009_SCI  "TT-7009 SCALED INPUT" %
%   F10:202  TT_7009_LOLO_SP  "TT-7009 LOLO ALARM SP" %
%   B3:0/1  ALARM_RESET  "ALARM RESET" %
%   T4:202  TT_7009_LOLO_DLY_TM  "TT-7009 LOLO ALARM DELAY" %
%   B3:19/14  "OSR" %
%   B3:19/15  "TT-7009 LOLO TRIGGER BIT" %

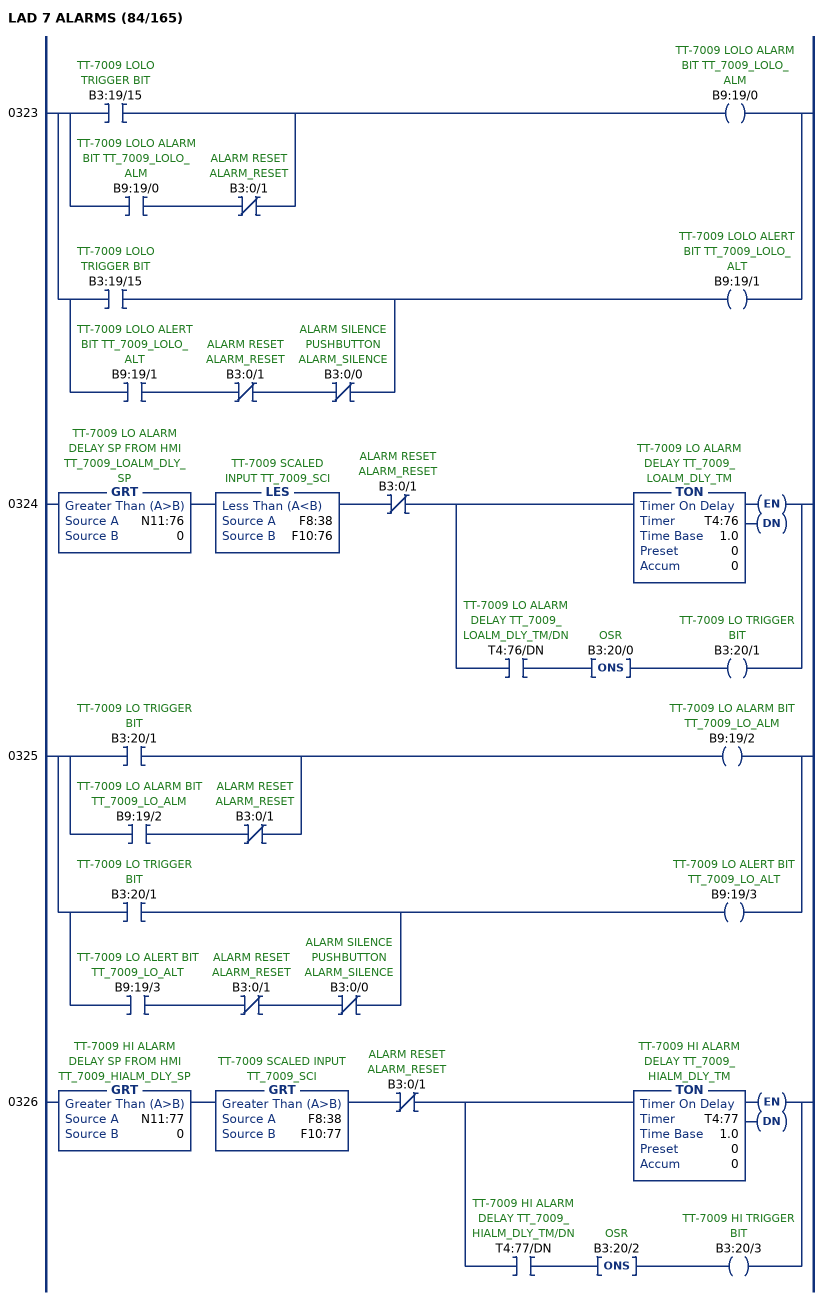
% Rung: 323 %
SOR BST BST XIC B3:19/15 NXB XIC B9:19/0 XIO B3:0/1 BND OTE B9:19/0 NXB BST XIC B3:19/15 NXB XIC B9:19/1 XIO B3:0/1 XIO B3:0/0 BND OTE B9:19/1 BND EOR
%   B3:19/15  "TT-7009 LOLO TRIGGER BIT" %
%   B9:19/0  TT_7009_LOLO_ALM  "TT-7009 LOLO ALARM BIT" %
%   B3:0/1  ALARM_RESET  "ALARM RESET" %
%   B9:19/1  TT_7009_LOLO_ALT  "TT-7009 LOLO ALERT BIT" %
%   B3:0/0  ALARM_SILENCE  "ALARM SILENCE PUSHBUTTON" %
% Rung: 324 %
SOR GRT N11:76 0 LES F8:38 F10:76 XIO B3:0/1 BST TON T4:76 1.0 0 0 NXB XIC T4:76/DN OSR B3:20/0 OTE B3:20/1 BND EOR
%   N11:76  TT_7009_LOALM_DLY_SP  "TT-7009 LO ALARM DELAY SP FROM HMI" %
%   F8:38  TT_7009_SCI  "TT-7009 SCALED INPUT" %
%   F10:76  TT_7009_LOALM_SP  "TT-7009 LO ALARM SP" %
%   B3:0/1  ALARM_RESET  "ALARM RESET" %
%   T4:76  TT_7009_LOALM_DLY_TM  "TT-7009 LO ALARM DELAY" %
%   B3:20/0  "OSR" %
%   B3:20/1  "TT-7009 LO TRIGGER BIT" %
% Rung: 325 %
SOR BST BST XIC B3:20/1 NXB XIC B9:19/2 XIO B3:0/1 BND OTE B9:19/2 NXB BST XIC B3:20/1 NXB XIC B9:19/3 XIO B3:0/1 XIO B3:0/0 BND OTE B9:19/3 BND EOR
%   B3:20/1  "TT-7009 LO TRIGGER BIT" %
%   B9:19/2  TT_7009_LO_ALM  "TT-7009 LO ALARM BIT" %
%   B3:0/1  ALARM_RESET  "ALARM RESET" %
%   B9:19/3  TT_7009_LO_ALT  "TT-7009 LO ALERT BIT" %
%   B3:0/0  ALARM_SILENCE  "ALARM SILENCE PUSHBUTTON" %
% Rung: 326 %
SOR GRT N11:77 0 GRT F8:38 F10:77 XIO B3:0/1 BST TON T4:77 1.0 0 0 NXB XIC T4:77/DN OSR B3:20/2 OTE B3:20/3 BND EOR
%   N11:77  TT_7009_HIALM_DLY_SP  "TT-7009 HI ALARM DELAY SP FROM HMI" %
%   F8:38  TT_7009_SCI  "TT-7009 SCALED INPUT" %
%   F10:77  TT_7009_HIALM_SP  "TT-7009 HI ALARM SP" %
%   B3:0/1  ALARM_RESET  "ALARM RESET" %
%   T4:77  TT_7009_HIALM_DLY_TM  "TT-7009 HI ALARM DELAY" %
%   B3:20/2  "OSR" %
%   B3:20/3  "TT-7009 HI TRIGGER BIT" %

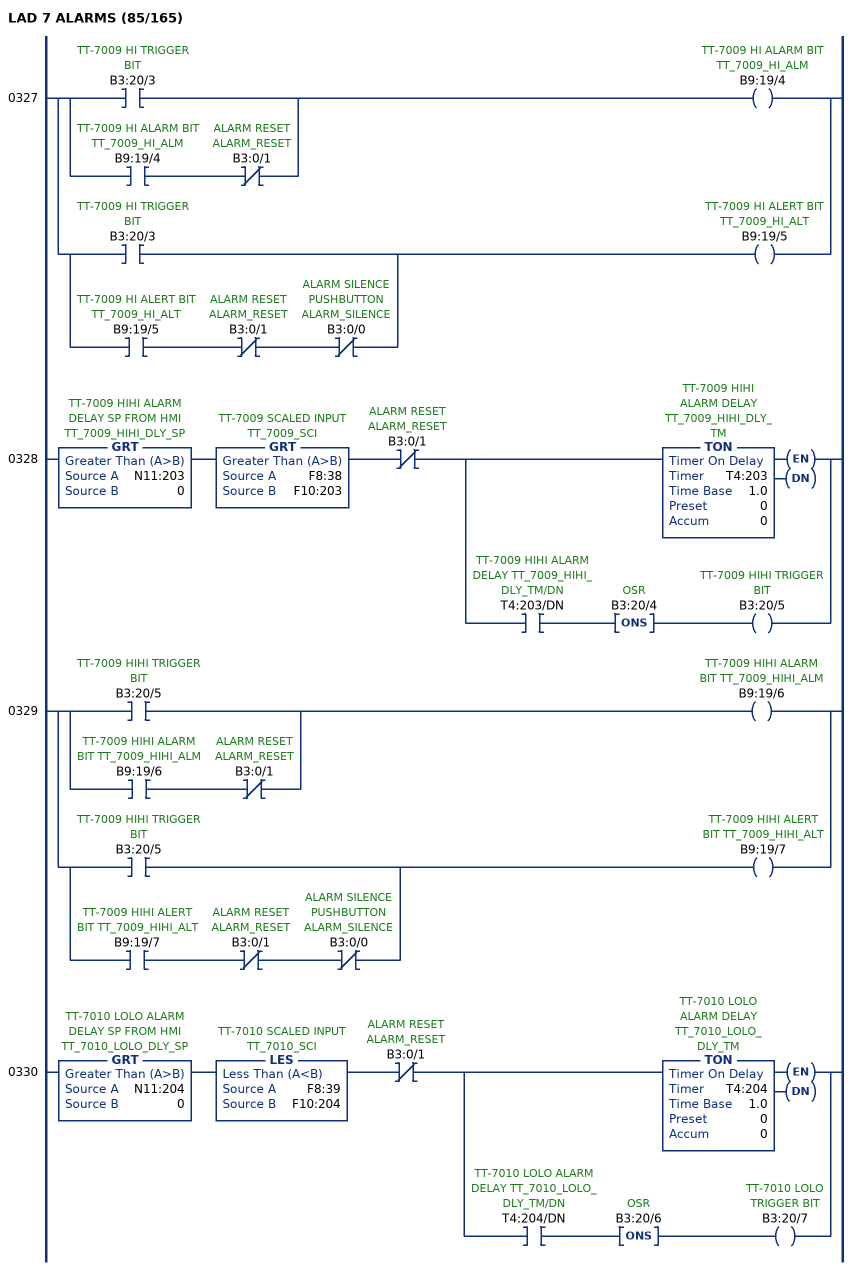
% Rung: 327 %
SOR BST BST XIC B3:20/3 NXB XIC B9:19/4 XIO B3:0/1 BND OTE B9:19/4 NXB BST XIC B3:20/3 NXB XIC B9:19/5 XIO B3:0/1 XIO B3:0/0 BND OTE B9:19/5 BND EOR
%   B3:20/3  "TT-7009 HI TRIGGER BIT" %
%   B9:19/4  TT_7009_HI_ALM  "TT-7009 HI ALARM BIT" %
%   B3:0/1  ALARM_RESET  "ALARM RESET" %
%   B9:19/5  TT_7009_HI_ALT  "TT-7009 HI ALERT BIT" %
%   B3:0/0  ALARM_SILENCE  "ALARM SILENCE PUSHBUTTON" %
% Rung: 328 %
SOR GRT N11:203 0 GRT F8:38 F10:203 XIO B3:0/1 BST TON T4:203 1.0 0 0 NXB XIC T4:203/DN OSR B3:20/4 OTE B3:20/5 BND EOR
%   N11:203  TT_7009_HIHI_DLY_SP  "TT-7009 HIHI ALARM DELAY SP FROM HMI" %
%   F8:38  TT_7009_SCI  "TT-7009 SCALED INPUT" %
%   F10:203  TT_7009_HIHI_SP  "TT-7009 HIHI ALARM SP" %
%   B3:0/1  ALARM_RESET  "ALARM RESET" %
%   T4:203  TT_7009_HIHI_DLY_TM  "TT-7009 HIHI ALARM DELAY" %
%   B3:20/4  "OSR" %
%   B3:20/5  "TT-7009 HIHI TRIGGER BIT" %
% Rung: 329 %
SOR BST BST XIC B3:20/5 NXB XIC B9:19/6 XIO B3:0/1 BND OTE B9:19/6 NXB BST XIC B3:20/5 NXB XIC B9:19/7 XIO B3:0/1 XIO B3:0/0 BND OTE B9:19/7 BND EOR
%   B3:20/5  "TT-7009 HIHI TRIGGER BIT" %
%   B9:19/6  TT_7009_HIHI_ALM  "TT-7009 HIHI ALARM BIT" %
%   B3:0/1  ALARM_RESET  "ALARM RESET" %
%   B9:19/7  TT_7009_HIHI_ALT  "TT-7009 HIHI ALERT BIT" %
%   B3:0/0  ALARM_SILENCE  "ALARM SILENCE PUSHBUTTON" %
% Rung: 330 %
SOR GRT N11:204 0 LES F8:39 F10:204 XIO B3:0/1 BST TON T4:204 1.0 0 0 NXB XIC T4:204/DN OSR B3:20/6 OTE B3:20/7 BND EOR
%   N11:204  TT_7010_LOLO_DLY_SP  "TT-7010 LOLO ALARM DELAY SP FROM HMI" %
%   F8:39  TT_7010_SCI  "TT-7010 SCALED INPUT" %
%   F10:204  TT_7010_LOLO_SP  "TT-7010 LOLO ALARM SP" %
%   B3:0/1  ALARM_RESET  "ALARM RESET" %
%   T4:204  TT_7010_LOLO_DLY_TM  "TT-7010 LOLO ALARM DELAY" %
%   B3:20/6  "OSR" %
%   B3:20/7  "TT-7010 LOLO TRIGGER BIT" %

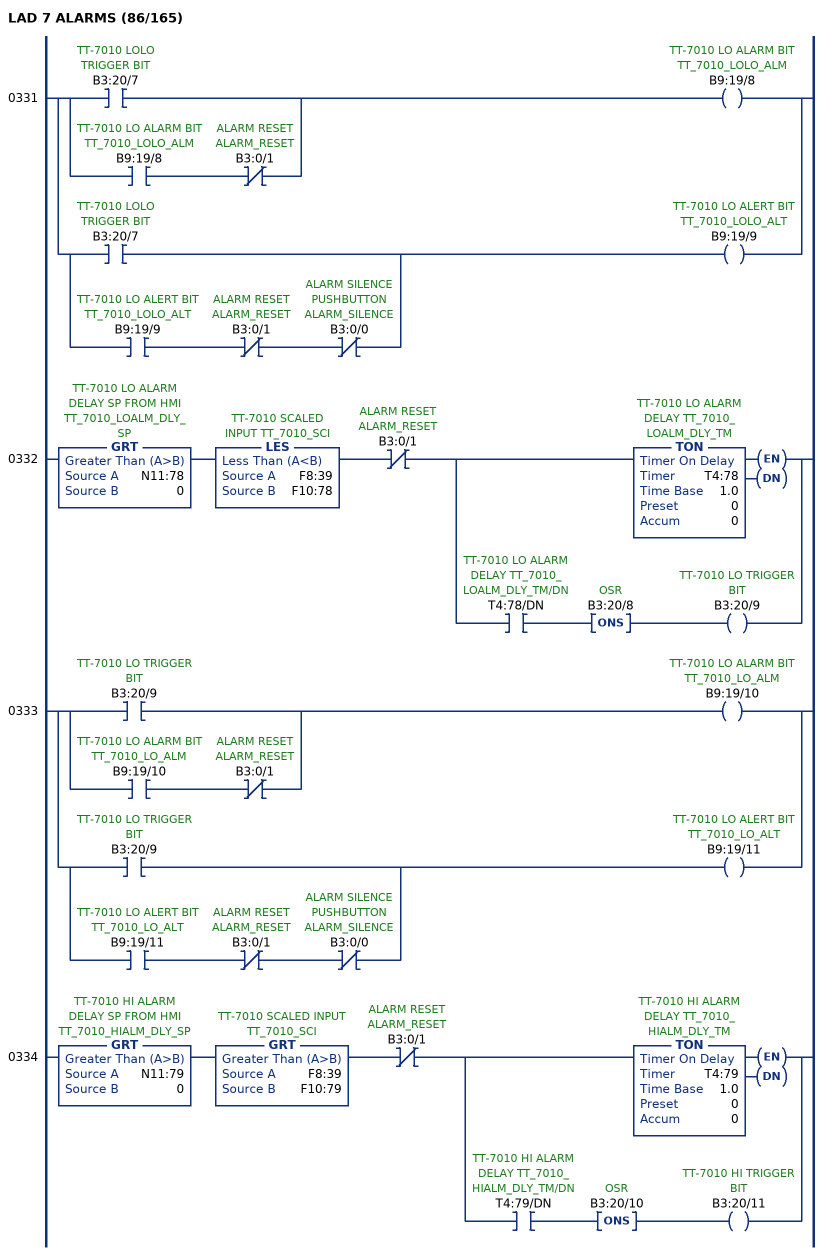
% Rung: 331 %
SOR BST BST XIC B3:20/7 NXB XIC B9:19/8 XIO B3:0/1 BND OTE B9:19/8 NXB BST XIC B3:20/7 NXB XIC B9:19/9 XIO B3:0/1 XIO B3:0/0 BND OTE B9:19/9 BND EOR
%   B3:20/7  "TT-7010 LOLO TRIGGER BIT" %
%   B9:19/8  TT_7010_LOLO_ALM  "TT-7010 LO ALARM BIT" %
%   B3:0/1  ALARM_RESET  "ALARM RESET" %
%   B9:19/9  TT_7010_LOLO_ALT  "TT-7010 LO ALERT BIT" %
%   B3:0/0  ALARM_SILENCE  "ALARM SILENCE PUSHBUTTON" %
% Rung: 332 %
SOR GRT N11:78 0 LES F8:39 F10:78 XIO B3:0/1 BST TON T4:78 1.0 0 0 NXB XIC T4:78/DN OSR B3:20/8 OTE B3:20/9 BND EOR
%   N11:78  TT_7010_LOALM_DLY_SP  "TT-7010 LO ALARM DELAY SP FROM HMI" %
%   F8:39  TT_7010_SCI  "TT-7010 SCALED INPUT" %
%   F10:78  TT_7010_LOALM_SP  "TT-7010 LO ALARM SP" %
%   B3:0/1  ALARM_RESET  "ALARM RESET" %
%   T4:78  TT_7010_LOALM_DLY_TM  "TT-7010 LO ALARM DELAY" %
%   B3:20/8  "OSR" %
%   B3:20/9  "TT-7010 LO TRIGGER BIT" %
% Rung: 333 %
SOR BST BST XIC B3:20/9 NXB XIC B9:19/10 XIO B3:0/1 BND OTE B9:19/10 NXB BST XIC B3:20/9 NXB XIC B9:19/11 XIO B3:0/1 XIO B3:0/0 BND OTE B9:19/11 BND EOR
%   B3:20/9  "TT-7010 LO TRIGGER BIT" %
%   B9:19/10  TT_7010_LO_ALM  "TT-7010 LO ALARM BIT" %
%   B3:0/1  ALARM_RESET  "ALARM RESET" %
%   B9:19/11  TT_7010_LO_ALT  "TT-7010 LO ALERT BIT" %
%   B3:0/0  ALARM_SILENCE  "ALARM SILENCE PUSHBUTTON" %
% Rung: 334 %
SOR GRT N11:79 0 GRT F8:39 F10:79 XIO B3:0/1 BST TON T4:79 1.0 0 0 NXB XIC T4:79/DN OSR B3:20/10 OTE B3:20/11 BND EOR
%   N11:79  TT_7010_HIALM_DLY_SP  "TT-7010 HI ALARM DELAY SP FROM HMI" %
%   F8:39  TT_7010_SCI  "TT-7010 SCALED INPUT" %
%   F10:79  TT_7010_HIALM_SP  "TT-7010 HI ALARM SP" %
%   B3:0/1  ALARM_RESET  "ALARM RESET" %
%   T4:79  TT_7010_HIALM_DLY_TM  "TT-7010 HI ALARM DELAY" %
%   B3:20/10  "OSR" %
%   B3:20/11  "TT-7010 HI TRIGGER BIT" %

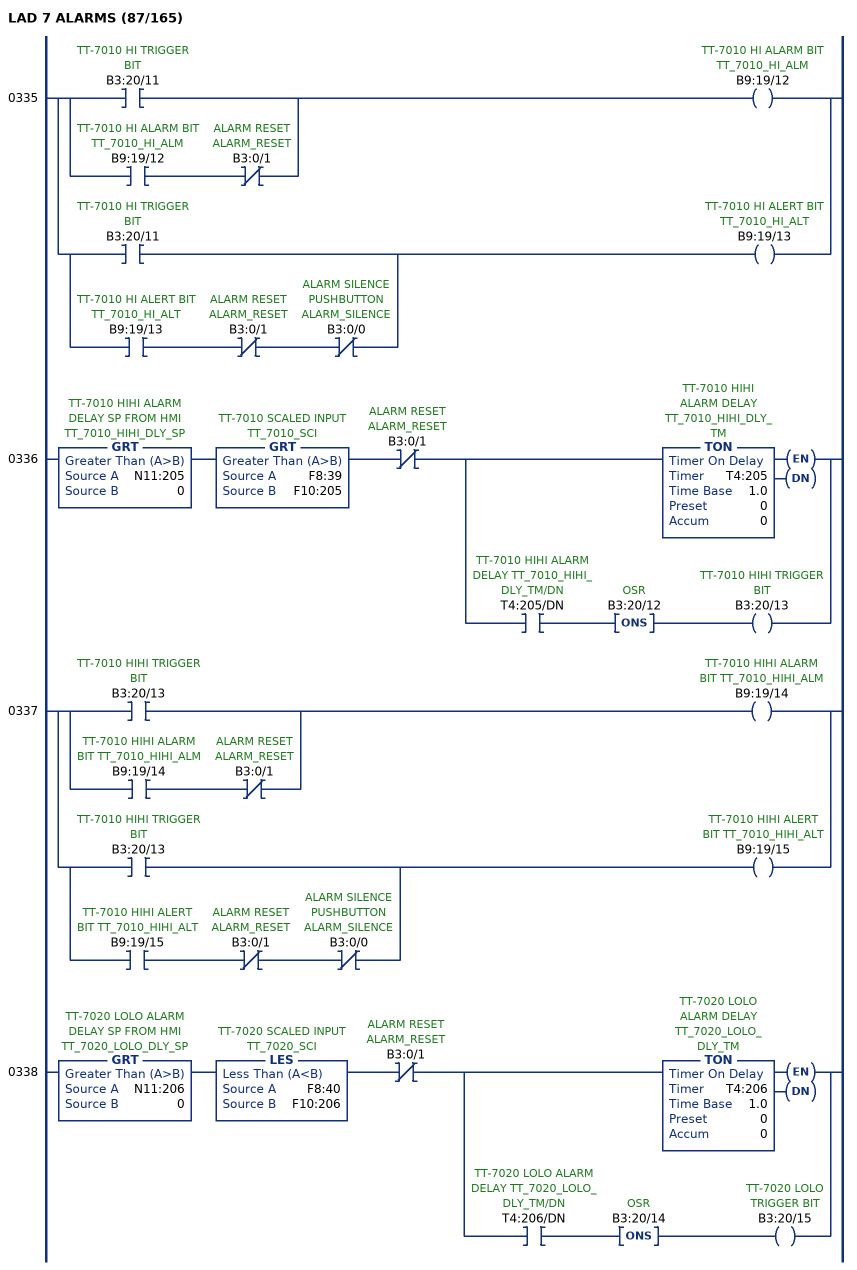
% Rung: 335 %
SOR BST BST XIC B3:20/11 NXB XIC B9:19/12 XIO B3:0/1 BND OTE B9:19/12 NXB BST XIC B3:20/11 NXB XIC B9:19/13 XIO B3:0/1 XIO B3:0/0 BND OTE B9:19/13 BND EOR
%   B3:20/11  "TT-7010 HI TRIGGER BIT" %
%   B9:19/12  TT_7010_HI_ALM  "TT-7010 HI ALARM BIT" %
%   B3:0/1  ALARM_RESET  "ALARM RESET" %
%   B9:19/13  TT_7010_HI_ALT  "TT-7010 HI ALERT BIT" %
%   B3:0/0  ALARM_SILENCE  "ALARM SILENCE PUSHBUTTON" %
% Rung: 336 %
SOR GRT N11:205 0 GRT F8:39 F10:205 XIO B3:0/1 BST TON T4:205 1.0 0 0 NXB XIC T4:205/DN OSR B3:20/12 OTE B3:20/13 BND EOR
%   N11:205  TT_7010_HIHI_DLY_SP  "TT-7010 HIHI ALARM DELAY SP FROM HMI" %
%   F8:39  TT_7010_SCI  "TT-7010 SCALED INPUT" %
%   F10:205  TT_7010_HIHI_SP  "TT-7010 HIHI ALARM SP" %
%   B3:0/1  ALARM_RESET  "ALARM RESET" %
%   T4:205  TT_7010_HIHI_DLY_TM  "TT-7010 HIHI ALARM DELAY" %
%   B3:20/12  "OSR" %
%   B3:20/13  "TT-7010 HIHI TRIGGER BIT" %
% Rung: 337 %
SOR BST BST XIC B3:20/13 NXB XIC B9:19/14 XIO B3:0/1 BND OTE B9:19/14 NXB BST XIC B3:20/13 NXB XIC B9:19/15 XIO B3:0/1 XIO B3:0/0 BND OTE B9:19/15 BND EOR
%   B3:20/13  "TT-7010 HIHI TRIGGER BIT" %
%   B9:19/14  TT_7010_HIHI_ALM  "TT-7010 HIHI ALARM BIT" %
%   B3:0/1  ALARM_RESET  "ALARM RESET" %
%   B9:19/15  TT_7010_HIHI_ALT  "TT-7010 HIHI ALERT BIT" %
%   B3:0/0  ALARM_SILENCE  "ALARM SILENCE PUSHBUTTON" %
% Rung: 338 %
SOR GRT N11:206 0 LES F8:40 F10:206 XIO B3:0/1 BST TON T4:206 1.0 0 0 NXB XIC T4:206/DN OSR B3:20/14 OTE B3:20/15 BND EOR
%   N11:206  TT_7020_LOLO_DLY_SP  "TT-7020 LOLO ALARM DELAY SP FROM HMI" %
%   F8:40  TT_7020_SCI  "TT-7020 SCALED INPUT" %
%   F10:206  TT_7020_LOLO_SP  "TT-7020 LOLO ALARM SP" %
%   B3:0/1  ALARM_RESET  "ALARM RESET" %
%   T4:206  TT_7020_LOLO_DLY_TM  "TT-7020 LOLO ALARM DELAY" %
%   B3:20/14  "OSR" %
%   B3:20/15  "TT-7020 LOLO TRIGGER BIT" %

